// TIA Portal V18 program export: 1 tag tables, 0 data types, 4 data blocks, 13 code blocks (in call order from the OBs), 40 instance data blocks

VAR_GLOBAL   // PLC tag table "Default tag table"
   Pulse1 AT %ID1000 : DInt;
   System_Byte AT %MB1 : Byte;
   FirstScan AT %M1.0 : Bool;
   DiagStatusUpdate AT %M1.1 : Bool;
   AlwaysTRUE AT %M1.2 : Bool;
   AlwaysFALSE AT %M1.3 : Bool;
   Clock_Byte AT %MB0 : Byte;
   Clock_10Hz AT %M0.0 : Bool;
   Clock_5Hz AT %M0.1 : Bool;
   "Clock_2.5Hz" AT %M0.2 : Bool;
   Clock_2Hz AT %M0.3 : Bool;
   "Clock_1.25Hz" AT %M0.4 : Bool;
   Clock_1Hz AT %M0.5 : Bool;
   "Clock_0.625Hz" AT %M0.6 : Bool;
   "Clock_0.5Hz" AT %M0.7 : Bool;
   Flowmeter_pulse AT %I0.0 : Bool;
   Simulate_pulse AT %Q0.4 : Bool;
   Date_time_trigger AT %M98.6 : Bool;
   PREV_Button AT %I1.3 : Bool;
   ENTER_Button AT %I1.4 : Bool;
   NEXT_Button AT %I1.5 : Bool;
   Pendant_START_Button AT %I0.3 : Bool;
   pendant_STOP_Button AT %I0.4 : Bool;
   emergency_mushroom AT %I0.1 : Bool;
   Capacitive_HLS AT %I0.5 : Bool;
   "in Loading" AT %M6.0 : Bool;
   stop_counting_up AT %M6.1 : Bool;
   "NEXT BUTTON FRONT" AT %M6.2 : Bool;
   "PREV BUTTON FRONT" AT %M6.3 : Bool;
   Pendant_emergency_stop AT %I0.2 : Bool;
   FCV_valve_closed AT %I0.6 : Bool;
   ESD_valve_closed AT %I0.7 : Bool;
   ESD_valve_open AT %I1.0 : Bool;
   Ground_monitor_IBC AT %I1.1 : Bool;
   Ground_monitor_truck AT %I1.2 : Bool;
   ESD_solenoid_valve AT %Q0.0 : Bool;
   To_contactor AT %Q0.3 : Bool;
   Flowmeter_analog AT %IW64 : Int;
   spare AT %IW1 : Int;
   "spare 0" AT %Q0.1 : Bool;
   "spare 1" AT %Q0.2 : Bool;
   drained_elapsed_time AT %MW8 : Int;
   RTD_PT100_1 AT %IW0 : Int;
   RTD_PT100_2 AT %IW4 : Int;
   RTD_PT100_3 AT %IW6 : Int;
   stop_counting_down AT %M6.4 : Bool;
END_VAR

DATA_BLOCK "Emergency_DB"   // DB22
{ S7_Optimized_Access := 'FALSE' }
VERSION : 0.1
// stored: AutoNumber true, IsOnlyStoredInLoadMemory false, IsWriteProtectedInAS false
   VAR
      Emergency_1 : Bool;
      Emergency_2 : Bool;
      Emergency_3 : Bool;
      Emergency_4 : Bool;
      Emergency_5 : Bool;
      Emergency_6 : Bool;
      Emergency_7 : Bool;
      Emergency_8 : Bool;
      Emergency_9 : Bool;
      Emergency_10 : Bool;
      Emergency_11 : Bool;
      Emergency_12 : Bool;
      Emergency_13 : Bool;
      Emergency_14 : Bool;
      Emergency_15 : Bool;
      Emergency_16 : Bool;
   END_VAR
BEGIN
END_DATA_BLOCK

DATA_BLOCK "HSC_variables"   // DB2
{ S7_Optimized_Access := 'TRUE' }
VERSION : 0.1
// stored: AutoNumber true, IsOnlyStoredInLoadMemory false, IsRetainMemResEnabled false, IsWriteProtectedInAS false, MemoryReserve 100
   VAR
      timer_drain_time : Time := T#2s;
   END_VAR
BEGIN
END_DATA_BLOCK

DATA_BLOCK "Var"   // DB1
{ S7_Optimized_Access := 'FALSE' }
VERSION : 0.1
// stored: AutoNumber true, IsOnlyStoredInLoadMemory false, IsWriteProtectedInAS false
   VAR RETAIN
      high_level_switch : Bool;
      panel_emergency_stop : Bool;
      pendant_emergency_stop : Bool;
      start_button : Bool;
      stop_button : Bool;
      FCV_valve_closed : Bool;
      FCV_valve_open : Bool;
      ESD_valve_closed : Bool;
      ESD_Valve_open : Bool;
      ground_signal1 : Bool;
      ground_signal2 : Bool;
      ESD_solenoid_valve_command : Bool;
      flowmeter_signal_Input : Int;
      flow_control_valve_output : Int;
      RTD_PT100_INPUT_1 : Int;
      RTD_PT100_INPUT_2 : Int;
      RTD_PT100_INPUT_3 : Int;
      Temperature : Int := 0;
      Temperature_threshold : Int := 100;
      Interlocks_idle : Bool;
      Grounding : Bool;
      In_loading : Bool;
      In_Draining : Bool;
      loaded_quantity : Real;
      Ready_to_Load : Bool;
      working_seq : Int;
      flow_meter_reset : Bool;
      "HSC_DATA.EdgeCount_real" : Real;
      "counter" : DInt;
      counter_real : Real;
      reset_counter : Bool;
      set_quantity : Int := 100;
      emergency_state : Bool;
      draining_flag : Bool;
      pump_signal : Bool;
      interlocks_loading : Bool;
      emergency_flag : Bool := false;
      instat_flowrate : Int;
      pause_flag : Bool;
      loading_flag : Bool;
      idle_flag : Bool;
      temperature_is_ok : Bool;
      drain_time_integer : Int := 10000;
      drain_time_time : Time := T#10000ms;
      drain_time_integer_seconds : Int := 10;
      Elapsed_drain_time : Int;
      Number_of_IBC : Int;
      Total_quantity : Real;
      lotto_terminato : Bool;
      freeze_counter : Bool;
      no_flow_states : Bool;
      FCV_low_flow_signal : Int := 5;
      FCV_high_flow_signal : Int := 10;
      quantity_of_LH_flow_intitial : Int := 20;
      quantity_of_LH_flow_percentage_initial : Int;
      quantity_of_HL_flow_final : Int := 20;
      quantity_of_HL_flow_percentage_final : Int;
      time_remained : Int;
      remained_quantity : Int;
      pulse_temp : DInt;
      recent_loaded_quantity : Int;
      No_of_IBC_all_time : Int;
   END_VAR
BEGIN
END_DATA_BLOCK

DATA_BLOCK "Var_HMI"   // DB10
{ S7_Optimized_Access := 'FALSE' }
VERSION : 0.1
// stored: AutoNumber true, IsOnlyStoredInLoadMemory false, IsWriteProtectedInAS false
   VAR
      "popup Emergency" : Bool;
      "popup warning" : Bool;
      Selector : UInt := 5;
      "page number" : UInt := 12;
      in_selection : Bool;
      emergency_popup : Bool;
      selection_no : Int;
      scrolling_1 : Int;
      scrolling_2 : Int;
   END_VAR
BEGIN
END_DATA_BLOCK

ORGANIZATION_BLOCK "Main"   // OB1, LAD, ProgramCycle
TITLE = "Main Program Sweep (Cycle)"
{ S7_Optimized_Access := 'TRUE' }
VERSION : 0.1
// stored: AutoNumber true, IsIECCheckEnabled false, SetENOAutomatically false
   VAR_INPUT
      Initial_Call : Bool;   // Initial call of this OB
      Remanence : Bool;   // =True, if remanent data are available
   END_VAR
BEGIN

REGION Network 1: Flow measurement
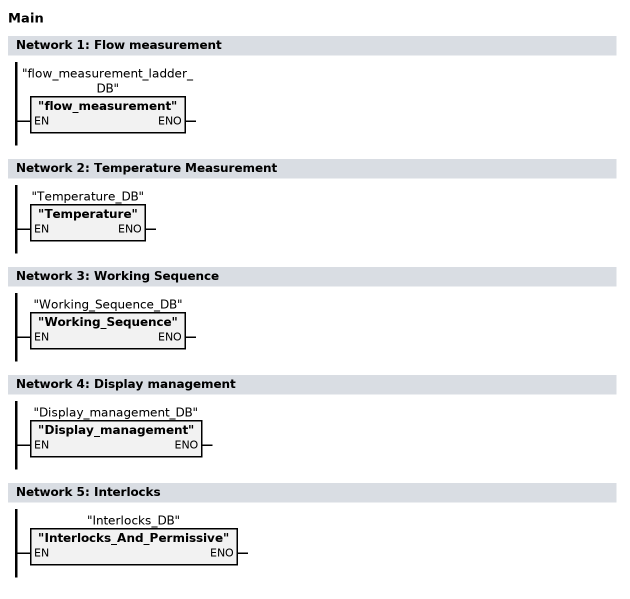
   RUNG wire#powerrail
      "flow_measurement_ladder_DB"()
   END_RUNG
   // the same network as SCL:
   "flow_measurement_ladder_DB"();   // "flow_measurement"
END_REGION

REGION Network 2: Temperature Measurement
   RUNG wire#powerrail
      "Temperature_DB"()
   END_RUNG
   // the same network as SCL:
   "Temperature_DB"();   // "Temperature"
END_REGION

REGION Network 3: Working Sequence
   RUNG wire#powerrail
      "Working_Sequence_DB"()
   END_RUNG
   // the same network as SCL:
   "Working_Sequence_DB"();   // "Working_Sequence"
END_REGION

REGION Network 4: Display management
   RUNG wire#powerrail
      "Display_management_DB"()
   END_RUNG
   // the same network as SCL:
   "Display_management_DB"();   // "Display_management"
END_REGION

REGION Network 5: Interlocks
   RUNG wire#powerrail
      "Interlocks_DB"()
   END_RUNG
   // the same network as SCL:
   "Interlocks_DB"();   // "Interlocks_And_Permissive"
END_REGION

REGION Network 6 (SCL): Emergency redundant signals
   // This is final command to ESD and the pump as a redundant command
   "To_contactor" := "To_contactor" AND "Var".emergency_state;
   "ESD_solenoid_valve" := "ESD_solenoid_valve" AND "Var".emergency_state;
END_REGION
END_ORGANIZATION_BLOCK

FUNCTION_BLOCK "flow_measurement"   // FB5, LAD
{ S7_Optimized_Access := 'TRUE' }
VERSION : 0.1
// stored: AutoNumber true, IsIECCheckEnabled false, IsRetainMemResEnabled false, MemoryReserve 100, SetENOAutomatically false, UDAEnableTagReadback false
   VAR
      K_factor : Real := 10.0;
   END_VAR
   VAR_TEMP
      Done : Bool;
      Busy : Bool;
      error : Bool;
      status : Word;
      pulse1_Temp : DInt;
      cv1 : Int;
   END_VAR
BEGIN

REGION Network 1: To simulate the Pulses from flow meter
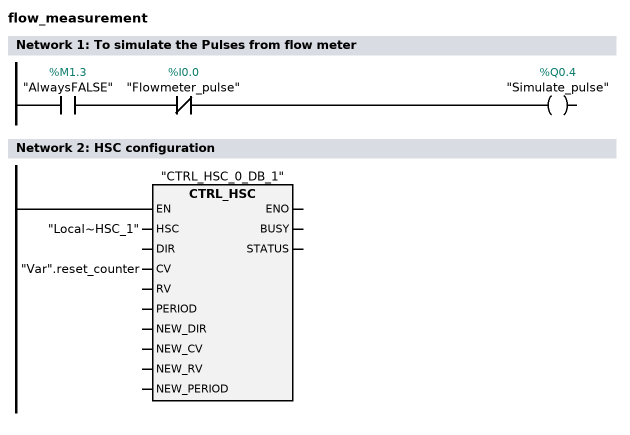
   RUNG wire#powerrail
      Contact( "AlwaysFALSE" )
      I_Contact( "Flowmeter_pulse" )
      Coil( "Simulate_pulse" )
   END_RUNG
   // the same network as SCL:
   "Simulate_pulse" := "AlwaysFALSE" AND NOT "Flowmeter_pulse";
END_REGION

REGION Network 2: HSC configuration
   RUNG wire#powerrail
      "CTRL_HSC_0_DB_1".CTRL_HSC(HSC := "Local~HSC_1", DIR :=, CV := "Var".reset_counter, RV :=, PERIOD :=, NEW_DIR :=, NEW_CV :=, NEW_RV :=, NEW_PERIOD :=, BUSY =>, STATUS =>)
   END_RUNG
   // the same network as SCL:
   "CTRL_HSC_0_DB_1"(HSC := "Local~HSC_1", CV := "Var".reset_counter);   // CTRL_HSC
END_REGION

REGION Network 3 (SCL): Read the value of the counter and put it in the Quantity value


   //counted pulse by HSC
   "Var".counter := "Pulse1";
   "Var".counter_real := DINT_TO_REAL(IN := "Var".counter);



   //K_factor should be edited correctly
   "Var".loaded_quantity := #K_factor * "Pulse1";



   //Time remained(in seconds, that's why multiplied by 3600)
   "Var".remained_quantity := ("Var".set_quantity - REAL_TO_INT("Var".loaded_quantity));
   "Var".time_remained := ("Var".remained_quantity / "Var".instat_flowrate) * 3600;
END_REGION

REGION Network 4 (SCL): Computing the recent loaded quantity (whenever pump starts)


   IF "Var".no_flow_states THEN
       "Var".pulse_temp := "Pulse1";
   END_IF;

   "Var".recent_loaded_quantity := ("Pulse1" - "Var".pulse_temp)* #K_factor;
END_REGION
END_FUNCTION_BLOCK

FUNCTION_BLOCK "Temperature"
{ S7_Optimized_Access := 'TRUE' }
VERSION : 0.1

BEGIN
	
	
	//A function of RTD1, RTD2, and RTD3 which the result gives the temperature. the following function needs modification
	"Var".Temperature := "Var".RTD_PT100_INPUT_1 + "Var".RTD_PT100_INPUT_2 + "Var".RTD_PT100_INPUT_3;
	
END_FUNCTION_BLOCK

FUNCTION_BLOCK "Working_Sequence"
{ S7_Optimized_Access := 'FALSE' }
VERSION : 0.1

BEGIN
	
	
	(* Explanation of variables and states
	    Working seq:
	         0  --> Idle
	        10 --> Loading
	        20 --> Emergency
	        25 --> Pause
	        
	*)
	
	REGION variable Assignation
	    
	    "Var".idle_flag := "Var".working_seq = 0;
	    "Var".loading_flag := "Var".working_seq = 10 OR "Var".working_seq = 11 OR "Var".working_seq = 12 OR "Var".working_seq = 13;
	    "Var".draining_flag := "Var".working_seq = 15;
	    "Var".emergency_flag := "Var".working_seq = 20;
	    "Var".pause_flag := "Var".working_seq = 25;
	    
	    
	    
	    "Rising_edge_start"(CLK := "Pendant_START_Button");
	    "Rising_edge_stop"(CLK := "pendant_STOP_Button");
	    "Rising_edge_enter"(CLK := "ENTER_Button");
	    "Rising_edge_next"(CLK := "NEXT_Button");
	    "Rising_edge_prev"(CLK := "PREV_Button");
	    
	    "Var".quantity_of_LH_flow_intitial := REAL_TO_INT("Var".quantity_of_LH_flow_percentage_initial * "Var".set_quantity / 100);
	    "Var".quantity_of_HL_flow_final := REAL_TO_INT("Var".quantity_of_HL_flow_percentage_final * "Var".set_quantity / 100);
	    
	END_REGION
	
	
	        
	        //Ready to load conditions (Interlocks + Quantity set + In loading )
	        IF  
	            "Var".In_loading  
	            AND "Var".set_quantity > 0   
	            AND "Var".Interlocks_idle
	        THEN
	            "Var".Ready_to_Load := 1;
	        ELSE
	            "Var".Ready_to_Load := 0;
	        END_IF;
	        
	        //IDLE state
	        IF "Var".working_seq = 0  THEN
	            
	            
	            
	            "ESD_solenoid_valve" := 0;
	            "Var".flow_control_valve_output := 0;
	            "To_contactor" := 0;
	            
	            // Go to emergency
	            IF NOT "Var".emergency_state THEN
	                
	                "Var".idle_flag := 0;
	                "Var".working_seq := 20;
	            END_IF;
	            
	            
	            
	            // Go to Loading    
	            IF      "Var".Ready_to_Load
	                AND "Var".interlocks_loading
	                AND "Var".In_loading
	                AND "Pendant_START_Button" 
	            THEN
	                
	                "Var".working_seq := 10;
	                
	                
	            END_IF;
	            
	            
	            // Go to Drain
	            IF      "Var".interlocks_loading
	                AND "Var".In_Draining
	                AND "Pendant_START_Button"
	                
	            THEN
	                
	                "Var".working_seq := 15;
	                
	            END_IF;
	            
	        END_IF;
	        
	        // Loading state
	        IF "Var".working_seq = 10 THEN
	            
	          
	            "To_contactor" := 1;
	            
	            "Flowmeter_pressure_timer".TON(IN := "Var".loading_flag,
	                                           PT := T#3000ms);
	            
	            //After 3 seconds open the valves (to reach to a certain pressure)
	            IF "Flowmeter_pressure_timer".Q THEN
	                
	                "Var".working_seq := 11;
	                
	            END_IF;
	            
	            
	        END_IF;
	        
	        //Low flow state, Initial
	        IF "Var".working_seq = 11 THEN
	            
	            //"To_contactor" := 1;
	            "Var".flow_control_valve_output := "Var".FCV_low_flow_signal;  // go to the value of low flow
	            "ESD_solenoid_valve" := 1;
	            
	            
	            // Going to High flow after loading of 50 kg, But not at the end of loading(in case of pause)
	            IF "Var".recent_loaded_quantity > "Var".quantity_of_LH_flow_intitial AND
	                "Var".remained_quantity>"Var".quantity_of_HL_flow_final
	            THEN
	                
	                "Var".working_seq := 12;
	                
	            END_IF;
	 
	        END_IF;
	        
	        //High flow state, Loading
	        IF "Var".working_seq = 12 THEN
	            
	            //Outputs in this state
	            //"To_contactor" := 1;
	            //"ESD_solenoid_valve" := 1;
	            "Var".flow_control_valve_output := "Var".FCV_high_flow_signal;
	            
	            
	            
	            // Going to final low flow, final
	            IF "Var".remained_quantity <= "Var".quantity_of_HL_flow_final  THEN
	                
	                "Var".working_seq := 13;
	                
	            END_IF;
	            
	
	            
	        END_IF;
	        
	        //Low flow state, final
	        IF "Var".working_seq = 13 THEN
	            
	         
	            "Var".flow_control_valve_output := "Var".FCV_low_flow_signal;  // go to the value of low flow
	            //"ESD_solenoid_valve" := 1;
	            //"To_contactor" := 1;
	            
	            
	            //condition for going out of this state are outside (like quantity reached, pause, emergency)
	            
	        END_IF;
	        
	        //Drain state
	        IF "Var".working_seq = 15 THEN
	            
	            
	                
	                // Outputs
	                "To_contactor" := 0;
	                "ESD_solenoid_valve" := 1;
	                "Var".flow_control_valve_output := "Var".FCV_high_flow_signal;
	                
	                
	                "Var".Elapsed_drain_time := TIME_TO_INT(IN := "IEC_Timer_0_DB_3".ET);
	                "Var".Elapsed_drain_time := ROUND("Var".Elapsed_drain_time / 1000);
	                
	                "IEC_Timer_0_DB_3".TON(IN := "Var".draining_flag,
	                                       PT := "Var".drain_time_time);
	                
	                
	                // Go to IDLE if the timer is reached   
	                IF "IEC_Timer_0_DB_3".Q THEN
	                    
	                    "Var".flow_control_valve_output := 0;
	                    "To_contactor" := 0;
	                    "ESD_solenoid_valve" := 0;
	                    
	                    "Var".In_Draining := 0;
	                    "Var".working_seq := 0;
	                    
	                    
	                    
	                    
	                END_IF;
	            END_IF;
	            
	        //Emergency state        
	        IF "Var".working_seq = 20 THEN
	            
	            
	            "To_contactor" := 0;
	            "ESD_solenoid_valve" := 0;
	            "Var".flow_control_valve_output := 0;
	           
	            // Go to Pause from emergency (when we are in loadinbg)
	            IF "Var".emergency_state AND "Rising_edge_enter".Q AND "Var".In_loading THEN
	                
	                "Rising_edge_enter".Q := 0;
	                "Var".working_seq := 25;
	                
	            END_IF;
	            
	            
	                // Go to Drain from emergency
	            IF "Var".emergency_state AND "Rising_edge_enter".Q AND "Var".In_Draining THEN
	                
	                
	                "Rising_edge_enter".Q := 0;
	                "Var".working_seq := 15;
	            END_IF;
	            
	            
	            
	            IF "Var".emergency_state AND "Rising_edge_enter".Q AND NOT "Var".In_loading THEN  //go to idle from Emergency
	                "Rising_edge_enter".Q := 0;
	                "Var".In_loading := 0;  
	                "Var".In_Draining := 0;
	                "Var".working_seq := 0;
	                
	            END_IF;
	            
	            
	            
	        END_IF;
	        
	        //Pause State   
	        IF "Var".working_seq = 25 THEN
	            
	            
	            
	            "To_contactor" := 0;
	            "ESD_solenoid_valve" := 0;
	            "Var".flow_control_valve_output := 0;
	            
	            //Go to IDLE from Loading
	            IF "Rising_edge_stop".Q AND "Var".In_loading  THEN
	                
	                "Rising_edge_stop".Q := 0;
	                "Var".Total_quantity := "Var".Total_quantity + "Var".loaded_quantity;
	                "Var".Number_of_IBC := "Var".Number_of_IBC + 1; // for the last partial IBC
	                "Var".In_loading := 0;
	                "IEC_Counter_0_DB".CV := 5;
	                "Var".lotto_terminato := 1;
	                "Var_HMI"."page number" := 15;
	                "Var".working_seq := 0;
	            END_IF;
	            
	            //Go to IDLE from Drain
	            IF "Rising_edge_stop".Q AND "Var".In_Draining THEN
	                
	                "Rising_edge_stop".Q := 0;
	                "Var".In_Draining := 0;
	                "IEC_Counter_0_DB".CV := 5;
	                "Var_HMI"."page number" := 12;
	                "Var".working_seq := 0;
	            END_IF;
	            
	            //Go to Draining    
	            IF "Var".In_Draining AND "Rising_edge_start".Q THEN
	                
	                "Rising_edge_start".Q := 0;
	                "Var".working_seq := 15;
	                
	                
	            END_IF;
	            
	            //Go to Loading
	            IF  "Var".In_loading AND  "Rising_edge_start".Q  THEN
	                
	                "Rising_edge_start".Q := 0;
	                "Var".working_seq := 10;
	                
	            END_IF;
	            
	            
	            
	        END_IF;
	        
	        
	        //*******************************************************************************************************
	        
	        //Go to Emergency if one emergency is lost
	        IF NOT "Var".emergency_state THEN
	            "Var".working_seq := 20;
	        END_IF;
	        
	        // Automatically turns off the pump and closes the valves (Go to IDLE)  
	        IF "Var".loaded_quantity >= "Var".set_quantity THEN
	            
	            "Var".In_loading := 0;
	            "Var".working_seq := 0;
	            
	        END_IF;
	        
	        //Going to pause mode, In loading value is not reset
	        IF "Rising_edge_stop".Q AND ("Var".In_loading OR "Var".In_Draining) THEN
	            
	            "Rising_edge_stop".Q := 0;
	            "Var".working_seq := 25;
	            
	        END_IF;
	        
	       
	        //Reseting the timers************************************************************************************
	        IF "Var".draining_flag =0 THEN
	            RESET_TIMER("IEC_Timer_0_DB_3");
	        END_IF;
	        
	        IF "Var".loading_flag = 0 THEN
	            RESET_TIMER("Flowmeter_pressure_timer");
	        END_IF;
	        //******************************************************************************************************
	        
	        
	        
	        
END_FUNCTION_BLOCK

FUNCTION_BLOCK "Display_management"   // FB7, LAD
{ S7_Optimized_Access := 'TRUE' }
VERSION : 0.1
// stored: AutoNumber true, IsIECCheckEnabled false, IsRetainMemResEnabled false, MemoryReserve 100, SetENOAutomatically false, UDAEnableTagReadback false
   VAR_TEMP   // added for the SCL form of the ladder/FBD networks
      _w1 : Bool;
      _w2 : Bool;
   END_VAR
BEGIN

REGION Network 1: reseting the Quantity, HSC
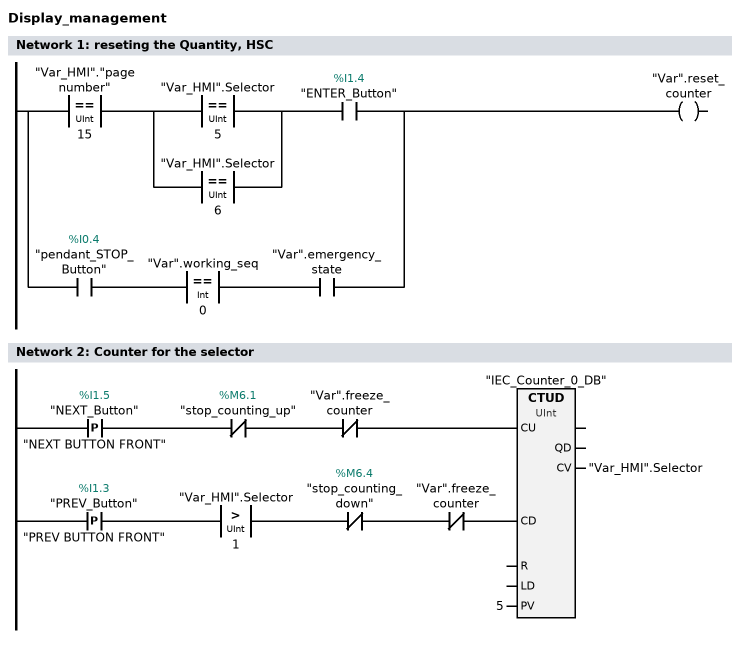
   RUNG wire#powerrail
      { S7_Templates := "SrcType := UInt" } EQ_Contact(in1 := "Var_HMI"."page number", in2 := 15)
      wire#w1
      { S7_Templates := "SrcType := UInt" } EQ_Contact(in1 := "Var_HMI".Selector, in2 := 5)
      wire#w2
      Contact( "ENTER_Button" )
      wire#w3
      Coil( "Var".reset_counter )
   END_RUNG
   RUNG wire#w1
      { S7_Templates := "SrcType := UInt" } EQ_Contact(in1 := "Var_HMI".Selector, in2 := 6)
   END_RUNG wire#w2
   RUNG wire#powerrail
      Contact( "pendant_STOP_Button" )
      { S7_Templates := "SrcType := Int" } EQ_Contact(in1 := "Var".working_seq, in2 := 0)
      Contact( "Var".emergency_state )
   END_RUNG wire#w3
   // the same network as SCL:
   "Var".reset_counter := (("Var_HMI"."page number" = 15) AND (("Var_HMI".Selector = 5) OR ("Var_HMI".Selector = 6)) AND "ENTER_Button") OR ("pendant_STOP_Button" AND ("Var".working_seq = 0) AND "Var".emergency_state);
END_REGION

REGION Network 2: Counter for the selector
   RUNG wire#powerrail
      P_Contact(operand := "NEXT_Button", bit := "NEXT BUTTON FRONT")
      I_Contact( "stop_counting_up" )
      I_Contact( "Var".freeze_counter )
      { S7_Templates := "value_type := UInt" } "IEC_Counter_0_DB".CTUD(cd := wire#w1, r :=, ld :=, pv := 5, qd =>, cv => "Var_HMI".Selector)
   END_RUNG
   RUNG wire#powerrail
      P_Contact(operand := "PREV_Button", bit := "PREV BUTTON FRONT")
      { S7_Templates := "SrcType := UInt" } GT_Contact(in1 := "Var_HMI".Selector, in2 := 1)
      I_Contact( "stop_counting_down" )
      I_Contact( "Var".freeze_counter )
   END_RUNG wire#w1
   // the same network as SCL:
   #_w1 := "NEXT_Button" AND NOT "NEXT BUTTON FRONT";   // rising edge of "NEXT_Button"
   "NEXT BUTTON FRONT" := "NEXT_Button";
   #_w2 := "PREV_Button" AND NOT "PREV BUTTON FRONT";   // rising edge of "PREV_Button"
   "PREV BUTTON FRONT" := "PREV_Button";
   "IEC_Counter_0_DB".CTUD(CU := #_w1 AND NOT "stop_counting_up" AND NOT "Var".freeze_counter,
                           CD := #_w2 AND ("Var_HMI".Selector > 1) AND NOT "stop_counting_down" AND NOT "Var".freeze_counter,
                           PV := 5,
                           CV => "Var_HMI".Selector);
END_REGION

REGION Network 3 (SCL): Condition for reseting the Menu counter
   IF     ("Var_HMI"."page number"=12 AND "Var_HMI".Selector>5)
       OR ("Var_HMI"."page number"=13 AND "Var_HMI".Selector>6)
       OR ("Var_HMI"."page number"=14 AND "Var_HMI".Selector>3)
       OR ("Var_HMI"."page number"=15 AND "Var_HMI".Selector>5)
       OR ("Var_HMI"."page number"=18 AND "Var_HMI".Selector>3)
       OR ("Var_HMI"."page number"=20 AND "Var_HMI".Selector>4)
       OR ("Var_HMI"."page number"=21 AND "Var_HMI".Selector>4)
       OR ("Var_HMI"."page number"=23 AND "Var_HMI".Selector>5)
       OR ("Var_HMI"."page number"=24 AND "Var_HMI".Selector>4)
       OR ("Var_HMI"."page number"=14 AND "Var_HMI".Selector>8)
       OR ("Var_HMI"."page number"=30 AND "Var_HMI".Selector>8)
       OR ("Var_HMI"."page number"=40 AND "Var_HMI".Selector>7)
   THEN
       "stop_counting_up" := 1;
   ELSE
       "stop_counting_up" := 0;
   END_IF;

   //Limitation for selector (OP fault prevetion)
   IF "Var_HMI"."page number" = 15 AND "Var_HMI".Selector<=5 THEN
       "stop_counting_down" := 1;
   ELSE
       "stop_counting_down" := 0;
   END_IF;


           // To freeze the counter
   "Var".freeze_counter := "Var".working_seq = 10
   OR "Var_HMI".in_selection
   OR "Var".emergency_flag
   OR "Var".pause_flag
   OR "Var".draining_flag
   OR ("Var_HMI"."page number" = 18);
END_REGION

REGION Network 4 (SCL): Page selector, for the Template icons

   //page12
   IF  "Var_HMI".Selector = 1 AND "Rising_edge_enter".Q THEN
       "Rising_edge_enter".Q := 0;
       "Var_HMI"."page number" := 12;
   END_IF;


   //page 20
   IF ("Var_HMI".Selector = 2 AND "Rising_edge_enter".Q) THEN
       "Rising_edge_enter".Q:= 0;
       "IEC_Counter_0_DB".CV := 5;
       "Var_HMI"."page number" := 20;

   END_IF;

   //page 20
   IF "Var_HMI"."page number" = 20 THEN

       IF "Var_HMI".Selector = 5 AND "Rising_edge_enter".Q THEN
           "IEC_Counter_0_DB".CV := 5;
           "Rising_edge_enter".Q:= 0;
           "Var_HMI"."page number" := 21;
       END_IF;

   END_IF;

   //page 21
   IF "Var_HMI"."page number" = 21 THEN

       IF "Var_HMI".Selector = 5 AND "Rising_edge_enter".Q THEN
           "Rising_edge_enter".Q := 0;
           "Var_HMI"."page number" := 20;
       END_IF;

   END_IF;

   //page 30
   IF ("Var_HMI".Selector = 3 AND "Rising_edge_enter".Q) THEN
       "Rising_edge_enter".Q := 0;
       "Var_HMI"."page number" := 30;
   END_IF;


   //page 40
   IF ("Var_HMI".Selector = 4 AND "Rising_edge_enter".Q) THEN
       "Rising_edge_enter".Q := 0;
       "Var_HMI"."page number" := 40;
   END_IF;
END_REGION

REGION Network 5 (SCL): Page 12, HOME
   //some condition should be added

   IF "Var_HMI"."page number" = 12 AND "Var".emergency_state THEN

       //Loading
       IF "Var_HMI".Selector = 5 AND "Rising_edge_enter".Q THEN

           "Var".Total_quantity := 0;
           "Var".lotto_terminato := 0;
           "Rising_edge_enter".Q := 0; 
           "IEC_Counter_0_DB".CV := 5;
           "Var_HMI"."page number" := 13;


       END_IF;

       //Drain
       IF "Var_HMI".Selector = 6 AND "Rising_edge_enter".Q THEN

           "Rising_edge_enter".Q := 0;
           "IEC_Counter_0_DB".CV := 6;
           "Var_HMI"."page number" := 23;


       END_IF;



   END_IF;
END_REGION

REGION Network 6 (SCL): Page 13 Loading setup
   //some condition should be added
   IF "Var_HMI"."page number" = 13 AND "Var".emergency_state THEN


       //"Var".reset_counter := 0;
       "EDIT_SET_QUANTITY".TON(IN:="ENTER_Button",
                               PT:=T#2000ms);

       //Set Timer for 
       IF "Var_HMI".Selector = 5 AND "EDIT_SET_QUANTITY".Q THEN

           "Var_HMI"."selection_no" := 1;
           "Var_HMI".in_selection:=1;


       END_IF;

       //Flow rate th
       IF "Var_HMI".Selector = 6 AND "EDIT_SET_QUANTITY".Q THEN

           "Var_HMI"."selection_no" := 2;
           "Var_HMI".in_selection := 1;

       END_IF;

       IF "Var_HMI".Selector=7 AND "Pendant_START_Button" AND "Var".set_quantity>0 AND "Var".FCV_high_flow_signal>0 THEN

           "Var".In_loading := 1;
           "Var".In_Draining := 0;
           "Var_HMI"."page number" := 14; 

       END_IF;

   END_IF;

   IF NOT "ENTER_Button" THEN
       RESET_TIMER("EDIT_SET_QUANTITY");
   END_IF;
END_REGION

REGION Network 7 (SCL): Page 14 In Loading
   //The condition need to be checked
   IF "Var_HMI"."page number" = 14 AND "Var".loaded_quantity >= "Var".set_quantity THEN
       "IEC_Counter_0_DB".CV := 5;
       "Var".Number_of_IBC := "Var".Number_of_IBC + 1;
       "Var".Total_quantity := "Var".Total_quantity + "Var".loaded_quantity;
       "Var_HMI"."page number" := 15;



   END_IF;
END_REGION

REGION Network 8 (SCL): Page 15, Lotto terminato
   IF "Var_HMI"."page number" = 15 AND "Var".emergency_state THEN



       "Var".lotto_terminato := 0;  //check this because you're resetting at page 12 

       IF "Var_HMI".Selector = 5 AND "Rising_edge_enter".Q THEN

           "Rising_edge_enter".Q := 0;
           "Var_HMI"."page number" := 13;

       END_IF;


       IF "Var_HMI".Selector = 6 AND "Rising_edge_enter".Q THEN

           "Rising_edge_enter".Q := 0;
           "IEC_Counter_0_DB".CV := 5;
           "Var_HMI"."page number" := 18;
           "Var".lotto_terminato := 1;

       END_IF;


   END_IF;
END_REGION

REGION Network 9 (SCL): Page 18, RIPIELOGO TERMINATO
   IF "Var_HMI"."page number"=18  THEN

       "Var".In_loading := 0;
       "Var".In_Draining := 0;


       IF "Rising_edge_enter".Q THEN
           "Var_HMI"."page number" := 12;
           "Var".Total_quantity := 0;
           "Rising_edge_enter".Q := 0;
           "Var".No_of_IBC_all_time := "Var".No_of_IBC_all_time + "Var".Number_of_IBC;
           "Var".Number_of_IBC := 0;
       END_IF;




   END_IF;
END_REGION

REGION Network 10 (SCL): Page 20 and 21, IOs
   IF "Var_HMI"."page number" = 20 THEN

       IF "Var_HMI".Selector = 5 AND "Rising_edge_enter".Q THEN
           "Var_HMI"."page number" := 21;
           "Rising_edge_enter".Q := 0;
       END_IF;

   END_IF;

   IF "Var_HMI"."page number" = 21 THEN

       IF "Var_HMI".Selector = 5 AND "Rising_edge_enter".Q THEN
           "Var_HMI"."page number" := 20;
           "Rising_edge_enter".Q := 0;
       END_IF;

   END_IF;
END_REGION

REGION Network 11 (SCL): Page 23, Drain pages setting
   IF "Var_HMI"."page number" = 23 AND "Var".emergency_state THEN


       "IEC_Timer_0_DB_4".TON(IN := "ENTER_Button",
                              PT := T#2S);




       //(Set Time FOR the timer, is it needed?
       IF "Var_HMI".Selector = 5 AND "IEC_Timer_0_DB_4".Q THEN

           "Var_HMI"."selection_no" := 3;
           "Var_HMI".in_selection := 1;

       END_IF;


       IF "Var_HMI".Selector = 6 AND "Pendant_START_Button" THEN
           "Var".In_Draining := 1;
           "Var_HMI"."page number" := 24;
           "IEC_Counter_0_DB".CV := 5;
       END_IF;


   END_IF;
END_REGION

REGION Network 12 (SCL): Page 24 Drain page
   IF "Var_HMI"."page number" = 24 THEN

       IF "Var_HMI".Selector = 5 AND "Rising_edge_enter".Q AND NOT ("Var".emergency_flag OR "Var".pause_flag OR "Var".draining_flag)  THEN

           "Var".In_Draining := 0;
           "Rising_edge_enter".Q := 0;
           "Var_HMI"."page number" := 12;
       END_IF;

   END_IF;
END_REGION

REGION Network 13 (SCL): Page 30, settings and default values


   IF "Var_HMI"."page number" = 30 THEN

       "IEC_Timer_0_DB_12".TON(IN:="ENTER_Button",
                               PT:=T#1500ms);




       IF "Var_HMI".Selector = 5 AND "IEC_Timer_0_DB_12".Q THEN
           "Var_HMI".selection_no := 8;
           "Var_HMI".in_selection := 1;


       END_IF;

       IF "Var_HMI".Selector = 6 AND "IEC_Timer_0_DB_12".Q THEN
           "Var_HMI".selection_no := 9;
           "Var_HMI".in_selection := 1;


       END_IF;

       IF "Var_HMI".Selector = 7 AND "IEC_Timer_0_DB_12".Q THEN
           "Var_HMI".selection_no := 10;
           "Var_HMI".in_selection := 1;


       END_IF;

       IF "Var_HMI".Selector = 8 AND "IEC_Timer_0_DB_12".Q THEN
           "Var_HMI".selection_no := 11;
           "Var_HMI".in_selection := 1;
           "Rising_edge_enter".Q := 0;

       END_IF;

       IF "Var_HMI".Selector = 9 AND "IEC_Timer_0_DB_12".Q THEN
           "Var_HMI".selection_no := 12;
           "Var_HMI".in_selection := 1;
           "Rising_edge_enter".Q := 0;
       END_IF;






   END_IF;

   IF NOT "ENTER_Button" THEN

       RESET_TIMER("IEC_Timer_0_DB_12");

   END_IF;
END_REGION

REGION Network 14 (SCL): page 40
   IF "Var_HMI"."page number" = 40 THEN

       "Scrolling_1_Timer".TON(IN := "ENTER_Button",
                               PT := T#1.5S);


       IF "Var_HMI".Selector = 5 AND "Scrolling_1_Timer".Q THEN

           "Var_HMI"."selection_no" := 4;
           "Var_HMI".in_selection := 1;


       END_IF;


       IF "Var_HMI".Selector = 6 AND "Scrolling_1_Timer".Q THEN

           "Var_HMI"."selection_no" := 5;
           "Var_HMI".in_selection := 1;

       END_IF;

      IF "Var_HMI".Selector = 7 AND "Scrolling_1_Timer".Q THEN

           "Var_HMI"."selection_no" := 6;
           "Var_HMI".in_selection := 1;

       END_IF;


       IF "Var_HMI".Selector = 8 AND "Scrolling_1_Timer".Q THEN

           "Var_HMI"."selection_no" := 7;
           "Var_HMI".in_selection := 1;
       END_IF;

   END_IF;
END_REGION

REGION Network 15 (SCL): In_Selection handling
   IF "Var_HMI".in_selection THEN

       CASE "Var_HMI".selection_no OF



           //Set Quantity       
           1:

                 "IEC_Timer_0_DB".TP(IN:="Clock_10Hz",
                                     PT:=T#0.001s);

                 IF "IEC_Timer_0_DB".Q THEN


                     IF "NEXT_Button" THEN
                         "Var".set_quantity := "Var".set_quantity + 10;
                     END_IF;


                     IF "PREV_Button" THEN
                         "Var".set_quantity := "Var".set_quantity - 10;
                         "Var".set_quantity := MAX(IN1 := "Var".set_quantity, IN2 := 0);


                     END_IF;


                     IF "ENTER_Button" THEN
                         "Var_HMI".in_selection := 0;
                         "Var_HMI".selection_no := 0;

                     END_IF;


                 END_IF;

                 ;





               //Set Flowrate
           2:

               "IEC_Timer_0_DB_1".TP(IN:="Clock_10Hz",
                                     PT:=T#0.001s);

               IF "IEC_Timer_0_DB_1".Q THEN


                   IF "NEXT_Button" THEN
                       "Var".FCV_high_flow_signal := "Var".FCV_high_flow_signal + 1;
                   END_IF;

                   IF "PREV_Button" THEN
                       "Var".FCV_high_flow_signal := "Var".FCV_high_flow_signal - 1;
                       "Var".FCV_high_flow_signal := MAX(IN1 := "Var".FCV_high_flow_signal, IN2 := 0);
                   END_IF;

                   IF "ENTER_Button" THEN
                       "Var_HMI".in_selection := 0;
                       "Var_HMI".selection_no := 0;
                   END_IF;

               END_IF;

               ;




               //Draining time
           3:


               "IEC_Timer_0_DB_2".TP(IN := "Clock_10Hz",
                                     PT := T#0.01s);

               IF "IEC_Timer_0_DB_2".Q THEN

                   IF "NEXT_Button" THEN
                       "Var".drain_time_integer := "Var".drain_time_integer + 100;
                       "Var".drain_time_integer_seconds := ROUND(IN := "Var".drain_time_integer / 1000);

                   END_IF;

                   IF "PREV_Button" THEN
                       "Var".drain_time_integer := "Var".drain_time_integer - 100;
                       "Var".drain_time_integer_seconds := ROUND(IN := "Var".drain_time_integer / 1000);
                       "Var".drain_time_integer_seconds := MAX(IN1 := "Var".drain_time_integer_seconds, IN2 := 0);
                       END_IF;

                   IF "ENTER_Button" THEN
                       "Var".drain_time_time := INT_TO_TIME(IN := "Var".drain_time_integer);
                       "Var_HMI"."in_selection" := 0;
                       "Var_HMI".selection_no := 0;
                   END_IF;


               END_IF;

               ;




               //scrolling 1
                   4:

                   "IEC_Timer_0_DB_6".TP(IN:="Clock_10Hz",
                                         PT:=T#0.001S);
                   IF NOT "ENTER_Button" THEN

                       "Scrolling_1_Timer".IN := FALSE;
                       "Var_HMI".in_selection := 0;
                       "Var_HMI".selection_no := 0;
                   END_IF;

                   IF "IEC_Timer_0_DB_6".Q AND "Var_HMI".in_selection  THEN

                       IF "ENTER_Button" THEN
                           "Var_HMI".scrolling_1 := "Var_HMI".scrolling_1 - 1;
                           "Var_HMI".scrolling_1 := MAX(IN1 := "Var_HMI".scrolling_1, IN2 := 0);
                       END_IF;

                   END_IF;

                   ;




                   //scrolling 2
           5:

               "IEC_Timer_0_DB_7".TP(IN := "Clock_10Hz",
                                     PT := T#0.001S);

               IF NOT "ENTER_Button" THEN

                   "Scrolling_1_Timer".IN := FALSE;
                   "Var_HMI".in_selection := 0;
                   "Var_HMI".selection_no := 0;
               END_IF;

               IF "IEC_Timer_0_DB_7".Q AND "Var_HMI".in_selection THEN

                   IF "ENTER_Button" THEN
                       "Var_HMI".scrolling_1 := "Var_HMI".scrolling_1 + 1;
                       "Var_HMI".scrolling_1 := MAX(IN1 := "Var_HMI".scrolling_1, IN2 := 0);
                   END_IF;

               END_IF;





               //scrolling 3
           6:

               "IEC_Timer_0_DB_8".TP(IN:="Clock_1Hz",
                                     PT:=T#0.001s);



               IF NOT "ENTER_Button" THEN

                   "Scrolling_1_Timer".IN := FALSE;
                   "Var_HMI".in_selection := 0;
                   "Var_HMI".selection_no := 0;
               END_IF;

               IF "IEC_Timer_0_DB_8".Q AND "Var_HMI".in_selection THEN

                   IF "ENTER_Button" THEN
                       "Var_HMI".scrolling_2 := "Var_HMI".scrolling_2 - 1;
                       "Var_HMI".scrolling_2 := MAX(IN1 := "Var_HMI".scrolling_2, IN2 := 0);
                   END_IF;

               END_IF;






               //scrolling 4 
           7:

               "IEC_Timer_0_DB_9".TP(IN:="Clock_1Hz",
                                     PT:=T#0.001s);



               IF NOT "ENTER_Button" THEN

                   "Scrolling_1_Timer".IN := FALSE;
                   "Var_HMI".in_selection := 0;
                   "Var_HMI".selection_no := 0;
               END_IF;

               IF "IEC_Timer_0_DB_9".Q AND "Var_HMI".in_selection THEN

                   IF "ENTER_Button" THEN
                       "Var_HMI".scrolling_2 := "Var_HMI".scrolling_2 + 1;
                   END_IF;

               END_IF;





               // Set the default Quantity
           8:

                  "IEC_Timer_0_DB_14".TP(IN:="Clock_10Hz",
                                         PT:=T#0.001s);
                  IF "IEC_Timer_0_DB_14".Q THEN

                  IF "NEXT_Button" THEN
                      "Var".set_quantity := "Var".set_quantity + 10;
                  END_IF;

                  IF "PREV_Button" THEN
                      "Var".set_quantity := "Var".set_quantity - 10;
                      "Var".set_quantity := MAX(IN1 := "Var".set_quantity, IN2 := 0);



                  END_IF;

                  IF "ENTER_Button" THEN
                      "Var_HMI".in_selection := 0;
                      "Var_HMI".selection_no := 0;


                  END_IF;
              END_IF;

               ;




               //Set the default flowrate
           9:
              "IEC_Timer_0_DB_17".TP(IN:="Clock_10Hz",
                                     PT:=T#0.001s);

              IF "IEC_Timer_0_DB_17".Q THEN

                  IF "NEXT_Button" THEN
                      "Var".FCV_high_flow_signal := "Var".FCV_high_flow_signal + 10;
                  END_IF;

                  IF "PREV_Button" THEN
                      "Var".FCV_high_flow_signal := "Var".FCV_high_flow_signal - 10;
                      "Var".FCV_high_flow_signal := MAX(IN1 := "Var".FCV_high_flow_signal, IN2 := 0);
                  END_IF;

                  IF "ENTER_Button" THEN

                      "Var_HMI".in_selection := 0;
                      "Var_HMI".selection_no := 0;


                  END_IF;

              END_IF;
               ;





               // Set default initial low flowrate percentage quantity
           10:


                   IF "Rising_edge_next".Q THEN
                       "Var".quantity_of_LH_flow_percentage_initial := "Var".quantity_of_LH_flow_percentage_initial + 1;
                       "Rising_edge_next".Q:=0;
                   END_IF;

                   IF "Rising_edge_prev".Q THEN
                       "Var".quantity_of_LH_flow_percentage_initial := "Var".quantity_of_LH_flow_percentage_initial - 1;
                       "Var".quantity_of_LH_flow_percentage_initial := MAX(IN1 := "Var".quantity_of_LH_flow_percentage_initial, IN2 := 0);
                       "Rising_edge_prev".Q := 0;

                   END_IF;

                   IF "Rising_edge_enter".Q THEN
                       "Var_HMI".in_selection := 0;
                       "Var_HMI".selection_no := 0;
                       "Rising_edge_enter".Q := 0;
                   END_IF;


               ;



               // Set default initial low flowrate percentage quantity
           11:

                   IF "Rising_edge_next".Q THEN
                       "Var".quantity_of_HL_flow_percentage_final := "Var".quantity_of_HL_flow_percentage_final + 1;
                       "Rising_edge_next".Q := 0;
                   END_IF;

                   IF "Rising_edge_prev".Q THEN
                       "Var".quantity_of_HL_flow_percentage_final := "Var".quantity_of_HL_flow_percentage_final - 1;
                       "Var".quantity_of_HL_flow_percentage_final := MAX(IN1 := "Var".quantity_of_HL_flow_percentage_final, IN2 := 0);
                       "Rising_edge_prev".Q := 0;
                   END_IF;

                   IF "Rising_edge_enter".Q THEN
                       "Var_HMI".in_selection := 0;
                       "Var_HMI".selection_no := 0;
                       "Rising_edge_enter".Q := 0;
                   END_IF;



               ;




               // Set default initial low flowrate percentage quantity
           12:
               "IEC_Timer_0_DB_16".TP(IN := "Clock_10Hz",
                                      PT := T#0.001S);
               IF "IEC_Timer_0_DB_16".Q THEN
                   IF "NEXT_Button" THEN
                       "Var".FCV_low_flow_signal:= "Var".FCV_low_flow_signal + 100;
                   END_IF;

                   IF "PREV_Button" THEN
                       "Var".FCV_low_flow_signal := "Var".FCV_low_flow_signal - 100;
                       "Var".FCV_low_flow_signal := MAX(IN1 := "Var".FCV_low_flow_signal, IN2 := 0);
                   END_IF;

                   IF "ENTER_Button" THEN
                       "Var_HMI".in_selection := 0;
                       "Var_HMI".selection_no := 0;

                   END_IF;

               END_IF;


               ;

       END_CASE;
   END_IF;
END_REGION

REGION Network 16 (SCL): Emergency Handling
   IF "Var".emergency_state AND "Var_HMI".emergency_popup AND "ENTER_Button" THEN

       "Var_HMI".emergency_popup := 0;

   END_IF;
END_REGION
END_FUNCTION_BLOCK

FUNCTION_BLOCK "Interlocks_And_Permissive"
{ S7_Optimized_Access := 'TRUE' }
VERSION : 0.1

BEGIN
	
	//High level,Pendant emergency stop, panel emergency Stop sensors are Normally close
	
	
	// Temperature
	"Var".temperature_is_ok := "Var".Temperature < "Var".Temperature_threshold;
	
	    //"Interlocks"
	    IF //"Capacitive_HLS"
	        //AND "Var".temperature_is_ok
	         "Var".emergency_state
	        //AND "FCV_valve_closed"
	        //AND "ESD_valve_closed"
	        //AND "Var".Grounding
	        
	        THEN
	        "Var".Interlocks_idle := 1;
	    ELSE
	        "Var".Interlocks_idle := 0;
	    END_IF;
	    
	    
	    
	    
	    
	    //Permissive (During the process)
	    IF  //"Capacitive_HLS"
	        //AND "Var".temperature_is_ok
	         "Var".emergency_state
	        //AND "Var".Grounding
	        
	    THEN
	        "Var".interlocks_loading := 1;
	    ELSE
	        "Var".interlocks_loading := 0;
	    END_IF;
	    
	
	
	    
END_FUNCTION_BLOCK

FUNCTION "Interlocks" : Void   // FC1, SCL
{ S7_Optimized_Access := 'TRUE' }
VERSION : 0.1
// stored: AutoNumber true, IsIECCheckEnabled false, SetENOAutomatically false, UDAEnableTagReadback false
   VAR_INPUT
      capacitive_HLS : Bool;
      temperature : Int;
      emergency_state : Bool;
      FCV_valve_closed : Bool;
      ESD_valve_closed : Bool;
      grounding : Bool;
      Temperature_threshold : Real;
   END_VAR
   VAR_OUTPUT
      temperature_is_ok : Bool;
      interlocks : Bool;
   END_VAR
BEGIN

   //High level,Pendant emergency stop, panel emergency Stop sensors are Normally close

   // Temperature, divided by ten because it the program it shows it 10x
   #temperature_is_ok := #temperature / 10 < #Temperature_threshold;

   //"Interlocks
   IF
       #temperature_is_ok
       AND #emergency_state
       AND #FCV_valve_closed
       AND #ESD_valve_closed
       AND #grounding
   THEN

       #interlocks := 1;
   ELSE
       #interlocks := 0;
   END_IF;
END_FUNCTION

ORGANIZATION_BLOCK "Emergency"   // OB31, LAD, CyclicInterrupt
{ S7_Optimized_Access := 'TRUE' }
VERSION : 0.1
// stored: AutoNumber true, IsIECCheckEnabled false, SetENOAutomatically false
   VAR_INPUT
      Initial_Call : Bool;   // Initial call of this OB
      Event_Count : Int;   // Events discarded
   END_VAR
BEGIN

REGION Network 1 (SCL): Checking ther conditions

   //1 FOR NO EMERGENCY, 0 IN CASE OF EMERGENCY
   //Only for the simulation, CAPACITIVE and PENDANT EMERGENCY should be added
   "Var".emergency_state := "emergency_mushroom";


   //Grounding is connected when it is 1 and 0 when it is not connected
   "Var".Grounding := "Ground_monitor_IBC" OR "Ground_monitor_truck";
END_REGION

REGION Network 2 (SCL): Defining kinds of unpredictable emergencies
   //Assign the emergencies

   // Emergency 1, fungo
   "Emergency_DB".Emergency_1 := NOT "emergency_mushroom";



   // Emergency 2, Pendant emergency
   "Emergency_DB".Emergency_2 := "Pendant_emergency_stop";



   // Emergency 3, Grounding
   "Emergency_DB".Emergency_3 := "Var".Grounding;



   // Emergency 4, HLS
   "Emergency_DB".Emergency_4 := "Capacitive_HLS";



   // Emergency 5, Temperature
   "Emergency_DB".Emergency_5 := NOT "Var".temperature_is_ok;



   // Emergency 6, NOT flow after 7 seconds OF In_loading state
   IF "Var".loading_flag THEN

       //signal of low flow, around 4mA, the value can be changed when we have connected the real FCV
       IF ABS("Flowmeter_analog" - 4) < 0.1 THEN

           //when it there is no flow, it starts a timer, if it remains the same for 7 seconds, shows an Emergency   
           "IEC_Timer_0_DB_5".TON(IN := "Var".loading_flag,
                                  PT := T#7S);



           IF "IEC_Timer_0_DB_5".Q THEN
               "Emergency_DB".Emergency_6 := 1;
           ELSE
               "Emergency_DB".Emergency_6 := 0;
           END_IF;

       END_IF;

   END_IF;
   // reseting the related timer
   IF NOT "Var".loading_flag THEN
       RESET_TIMER("IEC_Timer_0_DB_5"); 
   END_IF;



   "Var".no_flow_states := "Var".idle_flag OR "Var".emergency_flag OR "Var".pause_flag;
   // Emergency 7, Having flow in the idle Or pause state
   IF "Var".no_flow_states THEN

       "IEC_Timer_0_DB_11".TON(IN:="Var".no_flow_states,
                               PT:=T#3S);



       //If it is greater than the minimum (there is flow) after 3 seconds of being in Idle
       // the FLOW condition, can be changed! 
       IF "Flowmeter_analog" - 4 > 1 THEN


           IF "IEC_Timer_0_DB_11".Q THEN

               "Emergency_DB".Emergency_7 := 1;
           ELSE
               "Emergency_DB".Emergency_7 := 0;
           END_IF;


       END_IF;


   END_IF;
   //reseting the related timer
   IF NOT "Var".no_flow_states THEN
       RESET_TIMER("IEC_Timer_0_DB_11");
   END_IF;




   // Emergency 8, we are loading and FCV is closed
   IF "Var".loading_flag THEN

       //after 3 seconds being in loading and still the FCV is closed. 
       "IEC_Timer_0_DB_10".TON(IN:="Var".loading_flag,
                               PT:=T#3S);


       IF "IEC_Timer_0_DB_10".Q AND "FCV_valve_closed" THEN

           "Emergency_DB".Emergency_8 := 1;
       ELSE
           "Emergency_DB".Emergency_8 := 0;
       END_IF;

   END_IF;
   //reseting the timer in bellow



   // Emergency 9, we are in loading and ESD is closed
   IF "Var".loading_flag THEN

       //after 3 seconds being in loading and still the ESD is closed. 
       "IEC_Timer_0_DB_13".TON(IN := "Var".loading_flag,
                               PT := T#1500ms);




       IF "IEC_Timer_0_DB_13".Q AND "ESD_valve_closed" THEN

           "Emergency_DB".Emergency_9 := 1;
       ELSE
           "Emergency_DB".Emergency_9 := 0;
       END_IF;

   END_IF;
   //reseting the tiemrs
   IF NOT "Var".loading_flag THEN
       RESET_TIMER("IEC_Timer_0_DB_10");
       RESET_TIMER("IEC_Timer_0_DB_13");
   END_IF;
END_REGION
END_ORGANIZATION_BLOCK

ORGANIZATION_BLOCK "PID Control Valve"   // OB30, LAD, CyclicInterrupt
{ S7_Optimized_Access := 'TRUE' }
VERSION : 0.1
// stored: AutoNumber true, IsIECCheckEnabled false, SetENOAutomatically false
   VAR_INPUT
      Initial_Call : Bool;   // Initial call of this OB
      Event_Count : Int;   // Events discarded
   END_VAR
BEGIN

REGION Network 1: Put the variables for the pid
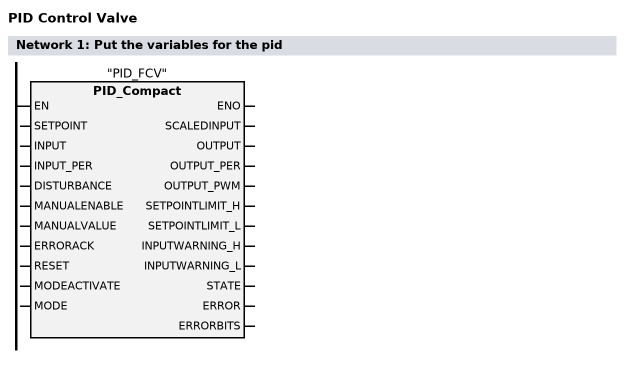
   RUNG wire#powerrail
      "PID_FCV".PID_Compact(Setpoint :=, Input :=, Input_PER :=, Disturbance :=, ManualEnable :=, ManualValue :=, ErrorAck :=, Reset :=, ModeActivate :=, Mode :=, ScaledInput =>, Output =>, Output_PER =>, Output_PWM =>, SetpointLimit_H =>, SetpointLimit_L =>, InputWarning_H =>, InputWarning_L =>, State =>, Error =>, ErrorBits =>)
   END_RUNG
   // the same network as SCL:
   "PID_FCV"();   // PID_Compact
END_REGION
END_ORGANIZATION_BLOCK

FUNCTION_BLOCK "Emergency_Block"   // FB3, SCL
{ S7_Optimized_Access := 'TRUE' }
VERSION : 0.1
// stored: AutoNumber true, IsIECCheckEnabled false, IsRetainMemResEnabled false, MemoryReserve 100, SetENOAutomatically false, UDAEnableTagReadback false
   VAR_OUTPUT
      emergency_state : Bool;
   END_VAR
BEGIN
   REGION Variables OF Emergency timers in Integer (TO show on HMI)
       "Var".Emer_timer_noFlow_int := TIME_TO_INT("Var".Emer_timer_noFlow);
       "Var".Emer_timer_Flow_int := TIME_TO_INT("Var".Emer_timer_Flow);
       "Var".Emer_timer_FCV_closed_int := TIME_TO_INT("Var".Emer_timer_FCV_closed);
       "Var".Emer_timer_ESD_closed_int := TIME_TO_INT("Var".Emer_timer_ESD_closed);
       "Var".Emer_timer_FCV_Open_int := TIME_TO_INT("Var".Emer_timer_FCV_Open);
       "Var".Emer_timer_ESD_Open_int := TIME_TO_INT("Var".Emer_timer_ESD_Open);
   END_REGION

   REGION Assign the emergencies


       // Emergency 1,*******************************************************************************************************
       REGION Emergency 1, fungo
           "Emergency_DB".Emergency_1 := NOT "emergency_mushroom";
       END_REGION

       // Emergency 2,*******************************************************************************************************
       REGION Emergency 2, pendant Emergency
           "Emergency_DB".Emergency_2 := NOT "pendant_emergency_stop";
       END_REGION

       // Emergency 3,*******************************************************************************************************
       REGION Emergency 3, Grounding
           "Emergency_DB".Emergency_3 := (NOT "ground_monitor_IBC") AND ("Var".loading_flag OR "Var".draining_flag);
       END_REGION

       // Emergency 4,*******************************************************************************************************
       REGION Emergency 4, High Level Switch
           "Emergency_DB".Emergency_4 := NOT "Capacitive_HLS";
       END_REGION

       // Emergency 5,*******************************************************************************************************
       REGION Emergency 5, Temperature
           "Emergency_DB".Emergency_5 := ("Temperature_RTD" / 10) > "Var".temperature_threshold AND "Temperature_RTD" < 29000;
       END_REGION

       // Emergency 6,******************************************************************************************************
       REGION Emergency 6, no flow in the loading state 
           IF "Var".loading_flag THEN

               "IEC_Timer_0_DB_5".TON(IN := "flowmeter_analog_feedback" < 1000,
                                      PT := "Var".Emer_timer_noFlow);

               IF "IEC_Timer_0_DB_5".Q THEN
                   "Emergency_DB".Emergency_6 := 1;
               END_IF;

           ELSE
               "Emergency_DB".Emergency_6 := 0;
           END_IF;

           IF NOT "Var".loading_flag OR "flowmeter_analog_feedback" > 1000 THEN
               RESET_TIMER("IEC_Timer_0_DB_5");
           END_IF;

       END_REGION

       // Emergency 7,******************************************************************************************************
       REGION Emergency 7, having flow in no flow state
           IF "Var".no_flow_states THEN

               "IEC_Timer_0_DB_11".TON(IN := "flowmeter_analog_feedback" > 50 AND "flowmeter_analog_feedback" < 29000,
                                       PT := "Var".Emer_timer_Flow);
               //If it is greater than the minimum (there is flow) after 3 seconds of being in Idle
               // the FLOW condition, can be changed!
               IF "IEC_Timer_0_DB_11".Q THEN
                   "Emergency_DB".Emergency_7 := 1;
               END_IF;
           END_IF;

           // reset its related timer 
           IF NOT ("flowmeter_analog_feedback" > 50 AND "flowmeter_analog_feedback" < 29000) OR NOT "Var".no_flow_states THEN

               "Emergency_DB".Emergency_7 := 0;
               RESET_TIMER("IEC_Timer_0_DB_11");
           END_IF;
       END_REGION

       // Emergency 8,*****************************************************************************************************
       REGION Emergency 8, FCV closed in loading
           IF "Var".loading_flag THEN

               //after 7 seconds being in loading and still the FCV is closed. 
               "IEC_Timer_0_DB_10".TON(IN := "FCV_valve_closed",
                                       PT := "Var".Emer_timer_FCV_closed);

               IF "IEC_Timer_0_DB_10".Q THEN
                   "Emergency_DB".Emergency_8 := 1;
               END_IF;
           ELSE
               "Emergency_DB".Emergency_8 := 0;
           END_IF;
           //resets the related timer 
           IF NOT "Var".loading_flag OR "FCV_valve_closed" THEN
               RESET_TIMER("IEC_Timer_0_DB_10");
           END_IF;
       END_REGION

       // Emergency 9,******************************************************************************************************
       REGION Emergency 9, ESD closed in loading
           IF "Var".loading_flag THEN
               //after 3 seconds being in loading and still the ESD is closed. 
               "IEC_Timer_0_DB_13".TON(IN := "ESD_valve_closed",
                                       PT := "Var".Emer_timer_ESD_closed);

               IF "IEC_Timer_0_DB_13".Q THEN

                   "Emergency_DB".Emergency_9 := 1;
               END_IF;
           END_IF;

           // If you are not in loading or ESD valve is not cloesed, this emergency should be reset.
           IF NOT "ESD_valve_closed" OR NOT "Var".loading_flag THEN
               RESET_TIMER("IEC_Timer_0_DB_13");
               "Emergency_DB".Emergency_9 := 0;
           END_IF;

       END_REGION

       //Emergency 10 **************************************************************************************************
       REGION Emergency 10, ESD open in no flow
           "IEC_Timer_0_DB".TON(IN := "Var".no_flow_states AND ("ESD_valve_open" OR NOT "ESD_valve_closed"),
                                PT := "Var".Emer_timer_ESD_Open);

           IF "IEC_Timer_0_DB".Q THEN
               "Emergency_DB".Emergency_10 := 1;
           END_IF;

           // Reseting the ESD valve Open timer
           IF NOT ("Var".no_flow_states AND ("ESD_valve_open" OR NOT "ESD_valve_closed")) THEN

               RESET_TIMER("IEC_Timer_0_DB");
               "Emergency_DB".Emergency_10 := 0;

           END_IF;
       END_REGION

       //Emergency 11 ***************************************************************************************************
       REGION emergency 11, FCV open in no flow

           "IEC_Timer_0_DB_1".TON(IN := "Var".no_flow_states AND ("FCV_valve_open" OR NOT "FCV_valve_closed"),
                                  PT := "Var".Emer_timer_FCV_Open);

           IF "IEC_Timer_0_DB_1".Q THEN
               "Emergency_DB".Emergency_11 := 1;
           END_IF;

           //reseting the FCV valve open timer
           IF NOT ("Var".no_flow_states AND ("FCV_valve_open" OR NOT "FCV_valve_closed")) THEN

               RESET_TIMER("IEC_Timer_0_DB_1");
               "Emergency_DB".Emergency_11 := 0;

           END_IF;
       END_REGION

       //Emergency 12,*****************************************************************************************************
       REGION Emergency 12, the cable OF flowmeter is disconnected


           //Flowmeter after 5 seconds of being disconnected, rises an alarm
           "IEC_Timer_0_DB_8".TON(IN:="flowmeter_analog_feedback" > 30000,
                                  PT:=T#10s);
           IF "IEC_Timer_0_DB_8".Q THEN
               "Emergency_DB".Emergency_12 := 1;
           END_IF;

           IF "flowmeter_analog_feedback" < 30000 THEN
               "Emergency_DB".Emergency_12 := 0;
               RESET_TIMER("IEC_Timer_0_DB_8");

           END_IF;


       END_REGION

       //Emergency 13******************************************************************************************************
       REGION Emergency 13, the cable OF RTD is disconnected

           //RTD after 5 seconds of being disconnected, rises an alarm

           "IEC_Timer_0_DB_7".TON(IN:="Temperature_RTD" > 30000,
                                  PT:=T#5s);
           IF "IEC_Timer_0_DB_7".Q THEN
               "Emergency_DB".Emergency_13 := 1;
           END_IF;


           IF "Temperature_RTD" < 30000 THEN
               "Emergency_DB".Emergency_13 := 0;
               RESET_TIMER("IEC_Timer_0_DB_7");
           END_IF;


       END_REGION

   END_REGION


   REGION Going TO Emergency
       //The #emergencies defined above
       #emergency_state := NOT (
       "Emergency_DB".Emergency_1
       OR "Emergency_DB".Emergency_2
       OR "Emergency_DB".Emergency_3 // Grounding only in flow state should be considered
       OR "Emergency_DB".Emergency_4
       OR "Emergency_DB".Emergency_5
       OR "Emergency_DB".Emergency_6
       OR "Emergency_DB".Emergency_7
       OR "Emergency_DB".Emergency_8
       OR "Emergency_DB".Emergency_9
       OR "Emergency_DB".Emergency_10
       OR "Emergency_DB".Emergency_11
       OR "Emergency_DB".Emergency_12
       OR "Emergency_DB".Emergency_13);

   END_REGION



   //1 FOR NO EMERGENCY, 0 IN CASE OF EMERGENCY
   // These are the flags only for the HMI pop up
   // To prevent from showing multiple emergencies on top, ELSIF is utilized
   REGION Emergency TO HMI
       //when there is an emergency, just set them immediately
       IF #emergency_state = 0 AND "Emergency_DB".Emergency_1 THEN 
           "Emergency_DB".Emergency_1_flag := "Emergency_DB".Emergency_1;

       ELSIF #emergency_state = 0 AND "Emergency_DB".Emergency_2 THEN
           "Emergency_DB".Emergency_2_flag := "Emergency_DB".Emergency_2;

       ELSIF #emergency_state = 0 AND "Emergency_DB".Emergency_3 THEN
           "Emergency_DB".Emergency_3_flag := "Emergency_DB".Emergency_3;

       ELSIF #emergency_state = 0 AND "Emergency_DB".Emergency_4 THEN
           "Emergency_DB".Emergency_4_flag := "Emergency_DB".Emergency_4;

       ELSIF #emergency_state = 0 AND "Emergency_DB".Emergency_5 THEN  
           "Emergency_DB".Emergency_5_flag := "Emergency_DB".Emergency_5;

       ELSIF #emergency_state = 0 AND "Emergency_DB".Emergency_6 THEN
           "Emergency_DB".Emergency_6_flag := "Emergency_DB".Emergency_6;

       ELSIF #emergency_state = 0 AND "Emergency_DB".Emergency_7 THEN
           "Emergency_DB".Emergency_7_flag := "Emergency_DB".Emergency_7;

       ELSIF #emergency_state = 0 AND "Emergency_DB".Emergency_8 THEN
           "Emergency_DB".Emergency_8_flag := "Emergency_DB".Emergency_8;

       ELSIF #emergency_state = 0 AND "Emergency_DB".Emergency_9 THEN
           "Emergency_DB".Emergency_9_flag := "Emergency_DB".Emergency_9;

       ELSIF #emergency_state = 0 AND "Emergency_DB".Emergency_10 THEN
           "Emergency_DB".Emergency_10_flag := "Emergency_DB".Emergency_10;

       ELSIF #emergency_state = 0 AND "Emergency_DB".Emergency_11 THEN
           "Emergency_DB".Emergency_11_flag := "Emergency_DB".Emergency_11;

       ELSIF #emergency_state = 0 AND "Emergency_DB".Emergency_12 THEN
           "Emergency_DB".Emergency_12_flag := "Emergency_DB".Emergency_12;

       ELSIF #emergency_state = 0 AND "Emergency_DB".Emergency_13 THEN
           "Emergency_DB".Emergency_13_flag := "Emergency_DB".Emergency_13;
       END_IF;

       // if the emergency is solved, then by pressing enter ,reset them
       IF "ENTER_Button" THEN
           "Emergency_DB".Emergency_1_flag  := "Emergency_DB".Emergency_1;
           "Emergency_DB".Emergency_2_flag  := "Emergency_DB".Emergency_2;
           "Emergency_DB".Emergency_3_flag  := "Emergency_DB".Emergency_3;
           "Emergency_DB".Emergency_4_flag  := "Emergency_DB".Emergency_4;
           "Emergency_DB".Emergency_5_flag  := "Emergency_DB".Emergency_5;
           "Emergency_DB".Emergency_6_flag  := "Emergency_DB".Emergency_6;
           "Emergency_DB".Emergency_7_flag  := "Emergency_DB".Emergency_7;
           "Emergency_DB".Emergency_8_flag  := "Emergency_DB".Emergency_8;
           "Emergency_DB".Emergency_9_flag  := "Emergency_DB".Emergency_9;
           "Emergency_DB".Emergency_10_flag := "Emergency_DB".Emergency_10;
           "Emergency_DB".Emergency_11_flag := "Emergency_DB".Emergency_11; 
           "Emergency_DB".Emergency_12_flag := "Emergency_DB".Emergency_12;
           "Emergency_DB".Emergency_13_flag := "Emergency_DB".Emergency_13;
           ;
       END_IF;
   END_REGION
END_FUNCTION_BLOCK

FUNCTION_BLOCK "HMI_In_selection_handling"   // FB4, SCL
{ S7_Optimized_Access := 'FALSE' }
VERSION : 0.1
// stored: AutoNumber true, IsIECCheckEnabled false, SetENOAutomatically false, UDAEnableTagReadback false
   VAR_INPUT
      step_size : Int := 50;
      Timer_duration : Time := T#1s;
      Time_pulse_speed : Time := T#1ms;
   END_VAR
   VAR_IN_OUT
      variable : Int;
   END_VAR
BEGIN


   IF "Rising_edge_next".Q THEN
       "Rising_edge_next".Q := 0;
       #variable := #variable + #step_size;
   END_IF;

   IF "Rising_edge_prev".Q THEN
       "Rising_edge_prev".Q := 0;
       #variable := #variable - #step_size;
       #variable := MAX(IN1 := #variable, IN2 := 0);
   END_IF;

   IF "Rising_edge_enter".Q THEN
       "Rising_edge_enter".Q := 0;
       "Var_HMI".in_selection := 0;
       "Var_HMI".selection_no := 0;

   END_IF;

   "IEC_Timer_0_DB_22".TON(IN:="NEXT_Button" OR "PREV_Button",
                           PT:=#Timer_duration);


   IF "IEC_Timer_0_DB_22".Q THEN


       "IEC_Timer_0_DB_16".TP(IN := "Clock_10Hz",
                              PT := #Time_pulse_speed);

       IF "IEC_Timer_0_DB_16".Q THEN

           IF "NEXT_Button" THEN
               #variable := #variable + 100;
           END_IF;

           IF "PREV_Button" THEN
               #variable := #variable - 100;
               #variable := MAX(IN1 := #variable, IN2 := 0);
           END_IF;

       END_IF;

       END_IF;


       IF NOT "NEXT_Button" AND NOT "PREV_Button" THEN
           RESET_TIMER("IEC_Timer_0_DB_22");
       END_IF;
END_FUNCTION_BLOCK

FUNCTION_BLOCK "Working_seq1"   // FB4, LAD
{ S7_Optimized_Access := 'TRUE' }
VERSION : 0.1
// stored: AutoNumber true, IsIECCheckEnabled false, IsRetainMemResEnabled false, MemoryReserve 100, SetENOAutomatically false, UDAEnableTagReadback false
BEGIN

REGION Network 2 (SCL)

   (* Explanation of variables and states
       Working seq:
            0  --> Idle
           10 --> Loading
           20 --> Emergency
           25 --> Pause

   *)


   //flags
   "Var".idle_flag := "Var".working_seq = 0;
   "Var".loading_flag := "Var".working_seq = 10 OR "Var".working_seq = 11 OR "Var".working_seq = 12 OR "Var".working_seq = 13;
   "Var".draining_flag := "Var".working_seq = 15;
   "Var".emergency_flag := "Var".working_seq = 20;
   "Var".pause_flag := "Var".working_seq = 25;



   "Rising_edge_start"(CLK := "Pendant_START_Button");
   "Rising_edge_stop"(CLK := "pendant_STOP_Button");
   "Rising_edge_enter"(CLK := "ENTER_Button");
   "Rising_edge_next"(CLK := "NEXT_Button");
   "Rising_edge_prev"(CLK := "PREV_Button");

   "Var".quantity_of_LH_flow_intitial := REAL_TO_INT("Var".quantity_of_LH_flow_percentage_initial * "Var".set_quantity / 100);
   "Var".quantity_of_HL_flow_final := REAL_TO_INT("Var".quantity_of_HL_flow_percentage_final * "Var".set_quantity / 100);



   //Ready to load conditions (Interlocks + Quantity set + In loading )
   IF
       "Var".In_loading
       AND "Var".set_quantity > 0
       AND "Var".Interlocks_idle
   THEN
       "Var".Ready_to_Load := 1;
   ELSE
       "Var".Ready_to_Load := 0;
   END_IF;


   //IDLE state
   IF "Var".working_seq = 0 THEN



       "ESD_solenoid_valve" := 0;
       "Var".flow_control_valve_output := 0;
       "To_contactor" := 0;

       // Go to emergency
       IF NOT "Var".emergency_state THEN

           "Var".idle_flag := 0;
           "Var".working_seq := 20;
       END_IF;



       // Go to Loading    
       IF "Var".Ready_to_Load
           AND "Var".interlocks_loading
           AND "Var".In_loading
           AND "Pendant_START_Button"
       THEN

           "Var".working_seq := 10;


       END_IF;


       // Go to Drain
       IF "Var".interlocks_loading
           AND "Var".In_Draining
           AND "Pendant_START_Button"

       THEN

           "Var".working_seq := 15;

       END_IF;

   END_IF;

   // Loading state
   IF "Var".working_seq = 10 THEN


       "To_contactor" := 1;

       "Flowmeter_pressure_timer".TON(IN := "Var".loading_flag,
                                      PT := T#3000ms);

       //After 3 seconds open the valves (to reach to a certain pressure)
       IF "Flowmeter_pressure_timer".Q THEN

           "Var".working_seq := 11;

       END_IF;


   END_IF;

   //Low flow state, Initial
   IF "Var".working_seq = 11 THEN

       //"To_contactor" := 1;
       "Var".flow_control_valve_output := "Var".FCV_low_flow_signal;  // go to the value of low flow
       "ESD_solenoid_valve" := 1;


       // Going to High flow after loading of 50 kg, But not at the end of loading(in case of pause)
       IF "Var".recent_loaded_quantity > "Var".quantity_of_LH_flow_intitial AND
           "Var".remained_quantity > "Var".quantity_of_HL_flow_final
       THEN

           "Var".working_seq := 12;

       END_IF;

   END_IF;

   //High flow state, Loading
   IF "Var".working_seq = 12 THEN

       //Outputs in this state
       //"To_contactor" := 1;
       //"ESD_solenoid_valve" := 1;
       "Var".flow_control_valve_output := "Var".FCV_high_flow_signal;



       // Going to final low flow, final
       IF "Var".remained_quantity <= "Var".quantity_of_HL_flow_final THEN

           "Var".working_seq := 13;

       END_IF;



   END_IF;

   //Low flow state, final
   IF "Var".working_seq = 13 THEN


       "Var".flow_control_valve_output := "Var".FCV_low_flow_signal;  // go to the value of low flow
       //"ESD_solenoid_valve" := 1;
       //"To_contactor" := 1;


       //condition for going out of this state are outside (like quantity reached, pause, emergency)

   END_IF;

   //Drain state
   IF "Var".working_seq = 15 THEN



       // Outputs
       "To_contactor" := 0;
       "ESD_solenoid_valve" := 1;
       "Var".flow_control_valve_output := "Var".FCV_high_flow_signal;


       "Var".Elapsed_drain_time := TIME_TO_INT(IN := "IEC_Timer_0_DB_3".ET);
       "Var".Elapsed_drain_time := ROUND("Var".Elapsed_drain_time / 1000);

       "IEC_Timer_0_DB_3".TON(IN := "Var".In_Draining,
                              PT := "Var".drain_time_time);


       // Go to IDLE if the timer is reached   
       IF "IEC_Timer_0_DB_3".Q THEN

           "Var".flow_control_valve_output := 0;
           "To_contactor" := 0;
           "ESD_solenoid_valve" := 0;

           "Var".In_Draining := 0;
           "Var".working_seq := 0;




       END_IF;
   END_IF;

   //Emergency state        
   IF "Var".working_seq = 20 THEN


       "To_contactor" := 0;
       "ESD_solenoid_valve" := 0;
       "Var".flow_control_valve_output := 0;

       // Go to Pause from emergency (when we are in loadinbg)
       IF "Var".emergency_state AND "Rising_edge_enter".Q AND "Var".In_loading THEN

           "Rising_edge_enter".Q := 0;
           "Var".working_seq := 25;

       END_IF;


       // Go to Drain from emergency
       IF "Var".emergency_state AND "Rising_edge_enter".Q AND "Var".In_Draining THEN


           "Rising_edge_enter".Q := 0;
           "Var".working_seq := 15;
       END_IF;



       IF "Var".emergency_state AND "Rising_edge_enter".Q AND NOT "Var".In_loading THEN  //go to idle from Emergency
           "Rising_edge_enter".Q := 0;
           "Var".In_loading := 0;
           "Var".In_Draining := 0;
           "Var".working_seq := 0;

       END_IF;



   END_IF;

   //Pause State   
   IF "Var".working_seq = 25 THEN



       "To_contactor" := 0;
       "ESD_solenoid_valve" := 0;
       "Var".flow_control_valve_output := 0;

       //Go to IDLE
       IF "Rising_edge_stop".Q THEN

           "Rising_edge_stop".Q := 0;
           "Var".Total_quantity := "Var".Total_quantity + "Var".loaded_quantity;
           "Var".Number_of_IBC := "Var".Number_of_IBC + 1; // for the last partial IBC
           "Var".In_loading := 0;
           "IEC_Counter_0_DB".CV := 5;
           "Var".lotto_terminato := 1;
           "Var_HMI"."page number" := 15;
           "Var".working_seq := 0;
       END_IF;


       //Go to Draining    
       IF "Var".In_Draining AND "Rising_edge_start".Q THEN

           "Rising_edge_start".Q := 0;
           "Var".working_seq := 15;


       END_IF;

       //Go to Loading
       IF "Var".In_loading AND "Rising_edge_start".Q THEN

           "Rising_edge_start".Q := 0;
           "Var".working_seq := 10;

       END_IF;



   END_IF;






   //*******************************************************************************************************

   //Go to Emergency if one emergency is lost
   IF NOT "Var".emergency_state THEN
       "Var".working_seq := 20;
   END_IF;

   // Automatically turns off the pump and closes the valves (Go to IDLE)  
   IF "Var".loaded_quantity >= "Var".set_quantity THEN

       "Var".In_loading := 0;
       "Var".working_seq := 0;

   END_IF;

   //Going to pause mode, In loading value is not reset
   IF "Rising_edge_stop".Q AND "Var".In_loading THEN

       "Rising_edge_stop".Q := 0;
       "Var".working_seq := 25;
   END_IF;


   //Reseting the timers************************************************************************************
   IF "Var".In_Draining = 0 THEN
       RESET_TIMER("IEC_Timer_0_DB_3");
   END_IF;

   IF "Var".In_loading = 0 THEN
       RESET_TIMER("Flowmeter_pressure_timer");
   END_IF;
   //******************************************************************************************************
END_REGION
END_FUNCTION_BLOCK

ORGANIZATION_BLOCK "Startup"
TITLE = "Complete Restart"
{ S7_Optimized_Access := 'TRUE' }
VERSION : 0.1

BEGIN
	
	
	"Var_HMI"."page number" := 12;
	
	
END_ORGANIZATION_BLOCK

DATA_BLOCK "Display_management_DB"   // DB17
VERSION : 0.1
// stored: AutoNumber true, InstanceOfName Display_management, InstanceOfType FB
"Display_management"
BEGIN
END_DATA_BLOCK

DATA_BLOCK "Emergency_Block_DB"   // DB2
VERSION : 0.1
// stored: AutoNumber true, InstanceOfName Emergency_Block, InstanceOfType FB
"Emergency_Block"
BEGIN
END_DATA_BLOCK

DATA_BLOCK "Interlocks_DB"   // DB3
VERSION : 0.1
// stored: AutoNumber true, InstanceOfName Interlocks_And_Permissive, InstanceOfType FB
"Interlocks_And_Permissive"
BEGIN
END_DATA_BLOCK

DATA_BLOCK "Temperature_DB"   // DB7
VERSION : 0.1
// stored: AutoNumber true, InstanceOfName Temperature, InstanceOfType FB
"Temperature"
BEGIN
END_DATA_BLOCK

DATA_BLOCK "Working_Sequence_DB"   // DB8
VERSION : 0.1
// stored: AutoNumber true, InstanceOfName Working_Sequence, InstanceOfType FB
"Working_Sequence"
BEGIN
END_DATA_BLOCK

DATA_BLOCK "flow_measurement_ladder_DB"   // DB5
VERSION : 0.1
// stored: AutoNumber true, InstanceOfName flow_measurement, InstanceOfType FB
"flow_measurement"
BEGIN
END_DATA_BLOCK

DATA_BLOCK "CTRL_HSC_0_DB_1"   // DB6
// stored: AutoNumber true, InstanceOfName CTRL_HSC, OfSystemLibElement CTRL_HSC, OfSystemLibVersion 1.0
"CTRL_HSC"
   // VAR_INPUT
   //    HSC : HW_HSC;
   //    DIR : Bool;
   //    CV : Bool;
   //    RV : Bool;
   //    PERIOD : Bool;
   //    NEW_DIR : Int;
   //    NEW_CV : DInt;
   //    NEW_RV : DInt;
   //    NEW_PERIOD : Int;
   // END_VAR
   // VAR_OUTPUT
   //    BUSY : Bool;
   //    STATUS : Word;
   // END_VAR
BEGIN
END_DATA_BLOCK

DATA_BLOCK "EDIT_SET_QUANTITY"   // DB16
{ S7_Optimized_Access := 'TRUE' }
// stored: AutoNumber true, InstanceOfName IEC_TIMER, OfSystemLibElement IEC_TIMER, OfSystemLibVersion 1.0
"IEC_TIMER"
   // VAR
   //    PT : Time;
   //    ET { ExternalWritable := 'False'} : Time;
   //    IN : Bool;
   //    Q { ExternalWritable := 'False'} : Bool;
   // END_VAR
BEGIN
END_DATA_BLOCK

DATA_BLOCK "Flowmeter_pressure_timer"   // DB18
{ S7_Optimized_Access := 'TRUE' }
// stored: AutoNumber true, InstanceOfName IEC_TIMER, OfSystemLibElement IEC_TIMER, OfSystemLibVersion 1.0
"IEC_TIMER"
   // VAR
   //    PT : Time;
   //    ET { ExternalWritable := 'False'} : Time;
   //    IN : Bool;
   //    Q { ExternalWritable := 'False'} : Bool;
   // END_VAR
BEGIN
END_DATA_BLOCK

DATA_BLOCK "IEC_Counter_0_DB"   // DB11
{ S7_Optimized_Access := 'TRUE' }
// stored: AutoNumber true, InstanceOfName IEC_UCOUNTER, OfSystemLibElement IEC_UCOUNTER, OfSystemLibVersion 1.0
"IEC_UCOUNTER"
   // VAR RETAIN
   //    CU : Bool;
   //    CD : Bool;
   //    R : Bool;
   //    LD : Bool;
   //    QU : Bool;
   //    QD : Bool;
   //    PV : UInt;
   //    CV : UInt;
   // END_VAR
BEGIN
END_DATA_BLOCK

DATA_BLOCK "IEC_Timer_0_DB"   // DB12
{ S7_Optimized_Access := 'TRUE' }
// stored: AutoNumber true, InstanceOfName IEC_TIMER, OfSystemLibElement IEC_TIMER, OfSystemLibVersion 1.0
"IEC_TIMER"
   // VAR
   //    PT : Time;
   //    ET { ExternalWritable := 'False'} : Time;
   //    IN : Bool;
   //    Q { ExternalWritable := 'False'} : Bool;
   // END_VAR
BEGIN
END_DATA_BLOCK

DATA_BLOCK "IEC_Timer_0_DB_1"   // DB13
{ S7_Optimized_Access := 'TRUE' }
// stored: AutoNumber true, InstanceOfName IEC_TIMER, OfSystemLibElement IEC_TIMER, OfSystemLibVersion 1.0
"IEC_TIMER"
   // VAR
   //    PT : Time;
   //    ET { ExternalWritable := 'False'} : Time;
   //    IN : Bool;
   //    Q { ExternalWritable := 'False'} : Bool;
   // END_VAR
BEGIN
END_DATA_BLOCK

DATA_BLOCK "IEC_Timer_0_DB_10"   // DB29
{ S7_Optimized_Access := 'TRUE' }
// stored: AutoNumber true, InstanceOfName IEC_TIMER, OfSystemLibElement IEC_TIMER, OfSystemLibVersion 1.0
"IEC_TIMER"
   // VAR
   //    PT : Time;
   //    ET { ExternalWritable := 'False'} : Time;
   //    IN : Bool;
   //    Q { ExternalWritable := 'False'} : Bool;
   // END_VAR
BEGIN
END_DATA_BLOCK

DATA_BLOCK "IEC_Timer_0_DB_11"   // DB30
{ S7_Optimized_Access := 'TRUE' }
// stored: AutoNumber true, InstanceOfName IEC_TIMER, OfSystemLibElement IEC_TIMER, OfSystemLibVersion 1.0
"IEC_TIMER"
   // VAR
   //    PT : Time;
   //    ET { ExternalWritable := 'False'} : Time;
   //    IN : Bool;
   //    Q { ExternalWritable := 'False'} : Bool;
   // END_VAR
BEGIN
END_DATA_BLOCK

DATA_BLOCK "IEC_Timer_0_DB_12"   // DB31
{ S7_Optimized_Access := 'TRUE' }
// stored: AutoNumber true, InstanceOfName IEC_TIMER, OfSystemLibElement IEC_TIMER, OfSystemLibVersion 1.0
"IEC_TIMER"
   // VAR
   //    PT : Time;
   //    ET { ExternalWritable := 'False'} : Time;
   //    IN : Bool;
   //    Q { ExternalWritable := 'False'} : Bool;
   // END_VAR
BEGIN
END_DATA_BLOCK

DATA_BLOCK "IEC_Timer_0_DB_13"   // DB32
{ S7_Optimized_Access := 'TRUE' }
// stored: AutoNumber true, InstanceOfName IEC_TIMER, OfSystemLibElement IEC_TIMER, OfSystemLibVersion 1.0
"IEC_TIMER"
   // VAR
   //    PT : Time;
   //    ET { ExternalWritable := 'False'} : Time;
   //    IN : Bool;
   //    Q { ExternalWritable := 'False'} : Bool;
   // END_VAR
BEGIN
END_DATA_BLOCK

DATA_BLOCK "IEC_Timer_0_DB_14"   // DB33
{ S7_Optimized_Access := 'TRUE' }
// stored: AutoNumber true, InstanceOfName IEC_TIMER, OfSystemLibElement IEC_TIMER, OfSystemLibVersion 1.0
"IEC_TIMER"
   // VAR
   //    PT : Time;
   //    ET { ExternalWritable := 'False'} : Time;
   //    IN : Bool;
   //    Q { ExternalWritable := 'False'} : Bool;
   // END_VAR
BEGIN
END_DATA_BLOCK

DATA_BLOCK "IEC_Timer_0_DB_15"   // DB34
{ S7_Optimized_Access := 'TRUE' }
// stored: AutoNumber true, InstanceOfName IEC_TIMER, OfSystemLibElement IEC_TIMER, OfSystemLibVersion 1.0
"IEC_TIMER"
   // VAR
   //    PT : Time;
   //    ET { ExternalWritable := 'False'} : Time;
   //    IN : Bool;
   //    Q { ExternalWritable := 'False'} : Bool;
   // END_VAR
BEGIN
END_DATA_BLOCK

DATA_BLOCK "IEC_Timer_0_DB_16"   // DB35
{ S7_Optimized_Access := 'TRUE' }
// stored: AutoNumber true, InstanceOfName IEC_TIMER, OfSystemLibElement IEC_TIMER, OfSystemLibVersion 1.0
"IEC_TIMER"
   // VAR
   //    PT : Time;
   //    ET { ExternalWritable := 'False'} : Time;
   //    IN : Bool;
   //    Q { ExternalWritable := 'False'} : Bool;
   // END_VAR
BEGIN
END_DATA_BLOCK

DATA_BLOCK "IEC_Timer_0_DB_17"   // DB36
{ S7_Optimized_Access := 'TRUE' }
// stored: AutoNumber true, InstanceOfName IEC_TIMER, OfSystemLibElement IEC_TIMER, OfSystemLibVersion 1.0
"IEC_TIMER"
   // VAR
   //    PT : Time;
   //    ET { ExternalWritable := 'False'} : Time;
   //    IN : Bool;
   //    Q { ExternalWritable := 'False'} : Bool;
   // END_VAR
BEGIN
END_DATA_BLOCK

DATA_BLOCK "IEC_Timer_0_DB_18"   // DB37
{ S7_Optimized_Access := 'TRUE' }
// stored: AutoNumber true, InstanceOfName IEC_TIMER, OfSystemLibElement IEC_TIMER, OfSystemLibVersion 1.0
"IEC_TIMER"
   // VAR
   //    PT : Time;
   //    ET { ExternalWritable := 'False'} : Time;
   //    IN : Bool;
   //    Q { ExternalWritable := 'False'} : Bool;
   // END_VAR
BEGIN
END_DATA_BLOCK

DATA_BLOCK "IEC_Timer_0_DB_19"   // DB40
{ S7_Optimized_Access := 'TRUE' }
// stored: AutoNumber true, InstanceOfName IEC_TIMER, OfSystemLibElement IEC_TIMER, OfSystemLibVersion 1.0
"IEC_TIMER"
   // VAR
   //    PT : Time;
   //    ET { ExternalWritable := 'False'} : Time;
   //    IN : Bool;
   //    Q { ExternalWritable := 'False'} : Bool;
   // END_VAR
BEGIN
END_DATA_BLOCK

DATA_BLOCK "IEC_Timer_0_DB_2"   // DB14
{ S7_Optimized_Access := 'TRUE' }
// stored: AutoNumber true, InstanceOfName IEC_TIMER, OfSystemLibElement IEC_TIMER, OfSystemLibVersion 1.0
"IEC_TIMER"
   // VAR
   //    PT : Time;
   //    ET { ExternalWritable := 'False'} : Time;
   //    IN : Bool;
   //    Q { ExternalWritable := 'False'} : Bool;
   // END_VAR
BEGIN
END_DATA_BLOCK

DATA_BLOCK "IEC_Timer_0_DB_20"   // DB41
{ S7_Optimized_Access := 'TRUE' }
// stored: AutoNumber true, InstanceOfName IEC_TIMER, OfSystemLibElement IEC_TIMER, OfSystemLibVersion 1.0
"IEC_TIMER"
   // VAR
   //    PT : Time;
   //    ET { ExternalWritable := 'False'} : Time;
   //    IN : Bool;
   //    Q { ExternalWritable := 'False'} : Bool;
   // END_VAR
BEGIN
END_DATA_BLOCK

DATA_BLOCK "IEC_Timer_0_DB_21"   // DB42
{ S7_Optimized_Access := 'TRUE' }
// stored: AutoNumber true, InstanceOfName IEC_TIMER, OfSystemLibElement IEC_TIMER, OfSystemLibVersion 1.0
"IEC_TIMER"
   // VAR
   //    PT : Time;
   //    ET { ExternalWritable := 'False'} : Time;
   //    IN : Bool;
   //    Q { ExternalWritable := 'False'} : Bool;
   // END_VAR
BEGIN
END_DATA_BLOCK

DATA_BLOCK "IEC_Timer_0_DB_22"   // DB43
{ S7_Optimized_Access := 'TRUE' }
// stored: AutoNumber true, InstanceOfName IEC_TIMER, OfSystemLibElement IEC_TIMER, OfSystemLibVersion 1.0
"IEC_TIMER"
   // VAR
   //    PT : Time;
   //    ET { ExternalWritable := 'False'} : Time;
   //    IN : Bool;
   //    Q { ExternalWritable := 'False'} : Bool;
   // END_VAR
BEGIN
END_DATA_BLOCK

DATA_BLOCK "IEC_Timer_0_DB_3"   // DB15
{ S7_Optimized_Access := 'TRUE' }
// stored: AutoNumber false, InstanceOfName IEC_TIMER, OfSystemLibElement IEC_TIMER, OfSystemLibVersion 1.0
"IEC_TIMER"
   // VAR
   //    PT : Time := T#0ms;
   //    ET { ExternalWritable := 'False'} : Time;
   //    IN : Bool;
   //    Q { ExternalWritable := 'False'} : Bool;
   // END_VAR
BEGIN
END_DATA_BLOCK

DATA_BLOCK "IEC_Timer_0_DB_4"   // DB19
{ S7_Optimized_Access := 'TRUE' }
// stored: AutoNumber true, InstanceOfName IEC_TIMER, OfSystemLibElement IEC_TIMER, OfSystemLibVersion 1.0
"IEC_TIMER"
   // VAR
   //    PT : Time;
   //    ET { ExternalWritable := 'False'} : Time;
   //    IN : Bool;
   //    Q { ExternalWritable := 'False'} : Bool;
   // END_VAR
BEGIN
END_DATA_BLOCK

DATA_BLOCK "IEC_Timer_0_DB_5"   // DB23
{ S7_Optimized_Access := 'TRUE' }
// stored: AutoNumber true, InstanceOfName IEC_TIMER, OfSystemLibElement IEC_TIMER, OfSystemLibVersion 1.0
"IEC_TIMER"
   // VAR
   //    PT : Time;
   //    ET { ExternalWritable := 'False'} : Time;
   //    IN : Bool;
   //    Q { ExternalWritable := 'False'} : Bool;
   // END_VAR
BEGIN
END_DATA_BLOCK

DATA_BLOCK "IEC_Timer_0_DB_6"   // DB25
{ S7_Optimized_Access := 'FALSE' }
// stored: AutoNumber true, InstanceOfName IEC_TIMER, OfSystemLibElement IEC_TIMER, OfSystemLibVersion 1.0
"IEC_TIMER"
   // VAR
   //    PT : Time;
   //    ET { ExternalWritable := 'False'} : Time;
   //    IN : Bool;
   //    Q { ExternalWritable := 'False'} : Bool;
   // END_VAR
BEGIN
END_DATA_BLOCK

DATA_BLOCK "IEC_Timer_0_DB_7"   // DB26
{ S7_Optimized_Access := 'FALSE' }
// stored: AutoNumber true, InstanceOfName IEC_TIMER, OfSystemLibElement IEC_TIMER, OfSystemLibVersion 1.0
"IEC_TIMER"
   // VAR
   //    PT : Time;
   //    ET { ExternalWritable := 'False'} : Time;
   //    IN : Bool;
   //    Q { ExternalWritable := 'False'} : Bool;
   // END_VAR
BEGIN
END_DATA_BLOCK

DATA_BLOCK "IEC_Timer_0_DB_8"   // DB27
{ S7_Optimized_Access := 'TRUE' }
// stored: AutoNumber true, InstanceOfName IEC_TIMER, OfSystemLibElement IEC_TIMER, OfSystemLibVersion 1.0
"IEC_TIMER"
   // VAR
   //    PT : Time;
   //    ET { ExternalWritable := 'False'} : Time;
   //    IN : Bool;
   //    Q { ExternalWritable := 'False'} : Bool;
   // END_VAR
BEGIN
END_DATA_BLOCK

DATA_BLOCK "IEC_Timer_0_DB_9"   // DB28
{ S7_Optimized_Access := 'TRUE' }
// stored: AutoNumber true, InstanceOfName IEC_TIMER, OfSystemLibElement IEC_TIMER, OfSystemLibVersion 1.0
"IEC_TIMER"
   // VAR
   //    PT : Time;
   //    ET { ExternalWritable := 'False'} : Time;
   //    IN : Bool;
   //    Q { ExternalWritable := 'False'} : Bool;
   // END_VAR
BEGIN
END_DATA_BLOCK

DATA_BLOCK "Rising_edge_enter"   // DB4
// stored: AutoNumber true, InstanceOfName R_TRIG, OfSystemLibElement R_TRIG, OfSystemLibVersion 1.0
"R_TRIG"
   // VAR_INPUT
   //    CLK : Bool;
   // END_VAR
   // VAR_OUTPUT
   //    Q : Bool;
   // END_VAR
   // VAR
   //    Stat_Bit : Bool;
   // END_VAR
BEGIN
END_DATA_BLOCK

DATA_BLOCK "Rising_edge_next"   // DB38
// stored: AutoNumber true, InstanceOfName R_TRIG, OfSystemLibElement R_TRIG, OfSystemLibVersion 1.0
"R_TRIG"
   // VAR_INPUT
   //    CLK : Bool;
   // END_VAR
   // VAR_OUTPUT
   //    Q : Bool;
   // END_VAR
   // VAR
   //    Stat_Bit : Bool;
   // END_VAR
BEGIN
END_DATA_BLOCK

DATA_BLOCK "Rising_edge_prev"   // DB39
// stored: AutoNumber true, InstanceOfName R_TRIG, OfSystemLibElement R_TRIG, OfSystemLibVersion 1.0
"R_TRIG"
   // VAR_INPUT
   //    CLK : Bool;
   // END_VAR
   // VAR_OUTPUT
   //    Q : Bool;
   // END_VAR
   // VAR
   //    Stat_Bit : Bool;
   // END_VAR
BEGIN
END_DATA_BLOCK

DATA_BLOCK "Rising_edge_start"   // DB20
// stored: AutoNumber true, InstanceOfName R_TRIG, OfSystemLibElement R_TRIG, OfSystemLibVersion 1.0
"R_TRIG"
   // VAR_INPUT
   //    CLK : Bool;
   // END_VAR
   // VAR_OUTPUT
   //    Q : Bool;
   // END_VAR
   // VAR
   //    Stat_Bit : Bool;
   // END_VAR
BEGIN
END_DATA_BLOCK

DATA_BLOCK "Rising_edge_stop"   // DB21
// stored: AutoNumber true, InstanceOfName R_TRIG, OfSystemLibElement R_TRIG, OfSystemLibVersion 1.0
"R_TRIG"
   // VAR_INPUT
   //    CLK : Bool;
   // END_VAR
   // VAR_OUTPUT
   //    Q : Bool;
   // END_VAR
   // VAR
   //    Stat_Bit : Bool;
   // END_VAR
BEGIN
END_DATA_BLOCK

DATA_BLOCK "Scrolling_1_Timer"   // DB24
{ S7_Optimized_Access := 'TRUE' }
// stored: AutoNumber true, InstanceOfName IEC_TIMER, OfSystemLibElement IEC_TIMER, OfSystemLibVersion 1.0
"IEC_TIMER"
   // VAR
   //    PT : Time;
   //    ET { ExternalWritable := 'False'} : Time;
   //    IN : Bool;
   //    Q { ExternalWritable := 'False'} : Bool;
   // END_VAR
BEGIN
END_DATA_BLOCK

DATA_BLOCK "PID_FCV"   // DB9
// stored: AutoNumber true, InstanceOfName PID_Compact, OfSystemLibElement PID_Compact, OfSystemLibVersion 2.3
PID_Compact   // technology object, version 2.3
   // VAR_INPUT
   //    Setpoint : Real;
   //    Input : Real;
   //    Input_PER : Int;
   //    Disturbance : Real;
   //    ManualEnable : Bool;
   //    ManualValue : Real;
   //    ErrorAck : Bool;
   //    Reset : Bool;
   //    ModeActivate : Bool;
   // END_VAR
   // VAR_OUTPUT
   //    ScaledInput { ExternalWritable := 'False'} : Real;
   //    Output { ExternalWritable := 'False'} : Real;
   //    Output_PER { ExternalWritable := 'False'} : Int;
   //    Output_PWM { ExternalWritable := 'False'} : Bool;
   //    SetpointLimit_H { ExternalWritable := 'False'} : Bool;
   //    SetpointLimit_L { ExternalWritable := 'False'} : Bool;
   //    InputWarning_H { ExternalWritable := 'False'} : Bool;
   //    InputWarning_L { ExternalWritable := 'False'} : Bool;
   //    State { ExternalWritable := 'False'} : Int;
   //    Error { ExternalWritable := 'False'} : Bool;
   //    ErrorBits { ExternalWritable := 'False'} : DWord;
   // END_VAR
   // VAR_IN_OUT
   //    Mode : Int;
   // END_VAR
   // VAR
   //    InternalDiagnostic : DWord;
   //    InternalVersion { ExternalWritable := 'False'} : DWord;
   //    InternalRTVersion : DWord;
   //    IntegralResetMode { S7_SetPoint := 'True'} : Int;
   //    OverwriteInitialOutputValue : Real;
   //    RunModeByStartup { S7_SetPoint := 'True'} : Bool;
   //    LoadBackUp : Bool;
   //    SetSubstituteOutput { S7_SetPoint := 'True'} : Bool;
   //    PhysicalUnit { ExternalWritable := 'False'; S7_SetPoint := 'True'} : Int;
   //    PhysicalQuantity { ExternalWritable := 'False'; S7_SetPoint := 'True'} : Int;
   //    ActivateRecoverMode { S7_SetPoint := 'True'} : Bool;
   // END_VAR
   // VAR RETAIN
   //    Warning { ExternalWritable := 'False'} : DWord;
   //    WarningInternal { ExternalWritable := 'False'} : DWord;
   // END_VAR
   // VAR
   //    Progress { ExternalWritable := 'False'} : Real;
   //    CurrentSetpoint { ExternalWritable := 'False'} : Real;
   //    CancelTuningLevel { S7_SetPoint := 'True'} : Real;
   //    SubstituteOutput { S7_SetPoint := 'True'} : Real;
   //    Config { S7_SetPoint := 'True'} : PID_CompactConfig;
   //    CycleTime { S7_SetPoint := 'True'} : PID_CycleTime;
   //    CtrlParamsBackUp { S7_SetPoint := 'True'} : PID_CompactControlParams;
   //    PIDSelfTune { S7_SetPoint := 'True'} : PID_CompactSelfTune;
   //    PIDCtrl { S7_SetPoint := 'True'} : PID_CompactControl;
   // END_VAR
   // VAR RETAIN
   //    Retain { S7_SetPoint := 'True'} : PID_CompactRetain;
   // END_VAR
BEGIN
END_DATA_BLOCK
